           20: //включаем ПИД ДВ (если режим работы от ПЧ)
               IF "DV_invertor_mode".Value THEN
                   IF "Control_DV".Mode = TRUE AND
                       "Control_DV".Mode_from_PLC = TRUE AND
                       "Control_DV".SP_PID = "RegMap".P_air_ventilation THEN
                       "Timer".VENTILATION_temp_IN := FALSE;
                       "Technology".Regim_ventilation_step := 22;
                   ELSE
                       "Control_DV".Mode := TRUE;
                       "Control_DV".Mode_from_PLC := TRUE;
                       "Control_DV".SP_PID := "RegMap".P_air_ventilation;
                       //переход на следующий шаг
                       "Timer".VENTILATION_temp_IN := FALSE;
                       "Technology".Regim_ventilation_step := 21;
                   END_IF;
               ELSE
                   "Control_DS".Mode_from_PLC := FALSE;
                   //переход через шаг (без ожидания)
                   "Timer".VENTILATION_temp_IN := FALSE;
                   "Technology".Regim_ventilation_step := 22;
               END_IF;

           21: //Ожидаем 6 сек
               "Timer".VENTILATION_temp_PT := T#6s;
               "Timer".VENTILATION_temp_IN := TRUE;
               //переход на следующий шаг
               IF "Timer".VENTILATION_temp_Q THEN
                   "Timer".VENTILATION_temp_IN := FALSE;
                   "Technology".Regim_ventilation_step := 22;
               END_IF;

           22: //Проверям достижение параметров вентиляции и удержание их в течении заданного времени
               "Timer".VENTILATION_temp_PT := T_CONV(INT_TO_DINT("Technology".SP_TIME_Ventilation_start) * 1000);
               "Timer".VENTILATION_temp_IN := "NAV_middle".Value AND     //НАВ достигли среднего положения
               NOT "NAD_close".Value AND  //НАД не закрыты
               "P_air_burner".Value > ("RegMap".P_air_ventilation * (100 - "Technology".DB_P_air_ventilation)) / 100 AND//Давление воздуха перед горелкой в норме
               (NOT "P_air_before_burner_min".Value OR "Protections_BLOCK".P_air_before_burner_min) AND
               //"Sensors".dP_furnace_boiler.Value > ("RegMap".dP_furnace_ventilation * (100 + "Technology".DB_dP_furnace_ventilation))/100 AND //Разряжение в норме
               "dP_furnace_boiler".Value < ("RegMap".dP_furnace_ventilation * (100 - "Technology".DB_dP_furnace_ventilation)) / 100 AND
               (NOT "dP_furnace_boiler_min".Value OR "Protections_BLOCK".dP_in_furnance_min);
               //переход на следующий шаг
               IF "Timer".VENTILATION_temp_Q THEN
                   "Timer".VENTILATION_temp_IN := FALSE;
                   "Timer".VENTILATION_IN := FALSE;
                   "Timer".VENTILATION_R := TRUE;
                   "Timer".VENTILATION_PT := T_CONV(INT_TO_DINT("Technology".SP_TIME_Ventilation) * 1000);
                   "Technology".Regim_ventilation_step := 23;
               END_IF;

           23: //ВЕНТИЛЯЦИЯ
               "Message".VENTILATION_run := "NAV_middle".Value AND     //НАВ достигли среднего положения
               NOT "NAD_close".Value AND  //НАД не закрыты
               "P_air_burner".Value > ("RegMap".P_air_ventilation * (100 - "Technology".DB_P_air_ventilation)) / 100 AND//Давление воздуха перед горелкой в норме
               (NOT "P_air_before_burner_min".Value OR "Protections_BLOCK".P_air_before_burner_min) AND
               //"Sensors".dP_furnace_boiler.Value > ("RegMap".dP_furnace_ventilation * (100 + "Technology".DB_dP_furnace_ventilation))/100 AND //Разряжение в норме
               "dP_furnace_boiler".Value < ("RegMap".dP_furnace_ventilation * (100 - "Technology".DB_dP_furnace_ventilation)) / 100 AND
               (NOT "dP_furnace_boiler_min".Value OR "Protections_BLOCK".dP_in_furnance_min);

               "Message".VENTILATION_not := NOT "Message".VENTILATION_run;

               "Message".VENTILATION_alarm := "Warning".P_air_before_burner_min OR "Warning".dP_furnace_boiler_min;

               //Запускаем таймер вентиляции (время задается уставкой) с контролем параметров:
               "Timer".VENTILATION_IN := "Message".VENTILATION_run;
               "Timer".VENTILATION_R := "Message".VENTILATION_alarm;
               "Timer".VENTILATION_PT := T_CONV(INT_TO_DINT("Technology".SP_TIME_Ventilation) * 1000);

               //Если таймер вентиляции вышел или если вентиляцию уже проводилась, то вентиляция успешно проведена
               IF "Timer".VENTILATION_Q OR "Technology".Ventilation_conducted THEN
                   "Timer".VENTILATION_IN := FALSE;
                   "Message".VENTILATION_run := FALSE;
                   "Message".VENTILATION_not := FALSE;
                   "Message".VENTILATION_alarm := FALSE;
                   "Message".VENTILATION_ok := TRUE;
                   "Technology".Ventilation_conducted := TRUE;
                   //переходим далее
                   "Technology".Regim_ventilation_step := 25;
                   "Technology".Test_press_run := FALSE;
                   "Technology".Test_ignition_run := FALSE;
               END_IF;
               //если вентиляция не выполнена, то переход на ожидание повторной вентиляции
               IF "Message".VENTILATION_alarm THEN
                   "Timer".VENTILATION_IN := FALSE;
                   "Message".VENTILATION_run := FALSE;
                   "Message".VENTILATION_not := FALSE;
                   "Technology".Regim_ventilation_step := 24;
               END_IF;

           24: //ожидание повторной команды при неудачной вентиляции 
               //повторная вентиляция
               IF "Btn_Ventilation".Value OR
                   "FRONT".Btn_Ventilation_HMI OR
                   "FRONT".Btn_Ventilation_SCADA THEN
                   "Message".VENTILATION_alarm := FALSE;
                   "Technology".Regim_ventilation_step := 0;
               END_IF;

           25: //ожидание выхода из вентиляции
               //взводим защиту Понижение давления воздуха перед горелкой
               "Alarm_Enable".P_air_before_burner_min := TRUE;
               //взводим защиту Понижение разряжения в топке
               "Alarm_Enable".dP_furnace_boiler_min := TRUE;
               //Если нажата кнопка РОЗЖИГ
               IF ("Btn_Ignition".Value OR "FRONT".Btn_Ignition_HMI OR "FRONT".Btn_Ignition_SCADA) THEN
                   //сброс розжиговых предупреждений    
                   "Warning".Not_flame_Igniter := FALSE;
                   "Warning".PZK2_not_open := FALSE;

                   IF //и все параматры вентиляци в норме
                       "NAV_middle".Value AND     //НАВ достигли среднего положения
                       NOT "NAD_close".Value AND  //НАД не закрыты
                       "P_air_burner".Value > ("RegMap".P_air_ventilation * (100 - "Technology".DB_P_air_ventilation)) / 100 AND//Давление воздуха перед горелкой в норме
                       (NOT "P_air_before_burner_min".Value OR "Protections_BLOCK".P_air_before_burner_min) AND
                       //"Sensors".dP_furnace_boiler.Value > ("RegMap".dP_furnace_ventilation * (100 + "Technology".DB_dP_furnace_ventilation))/100 AND //Разряжение в норме
                       "dP_furnace_boiler".Value < ("RegMap".dP_furnace_ventilation * (100 - "Technology".DB_dP_furnace_ventilation)) / 100 AND
                       (NOT "dP_furnace_boiler_min".Value OR "Protections_BLOCK".dP_in_furnance_min) THEN
                       "Message".VENTILATION_Check_param := FALSE;
                       "Message".VENTILATION_ok := FALSE;
                       //переход на ОПРЕССОВКА
                       "Technology".Regim := 4;
                   ELSE
                       "Message".VENTILATION_Check_param := TRUE;
                   END_IF;
               END_IF;

               //переход на ТЕСТОВУЮ ОПРЕССОВКУ по нажатию на кн.ТЕСТОВАЯ ОПРЕССОВКА
               IF "FRONT".Btn_test_press_HMI THEN
                   //сброс розжиговых предупреждений    
                   "Warning".Not_flame_Igniter := FALSE;
                   "Warning".PZK2_not_open := FALSE;

                   IF //и все параматры вентиляци в норме
                       "NAV_middle".Value AND     //НАВ достигли среднего положения
                       NOT "NAD_close".Value AND  //НАД не закрыты
                       "P_air_burner".Value > ("RegMap".P_air_ventilation * (100 - "Technology".DB_P_air_ventilation)) / 100 AND//Давление воздуха перед горелкой в норме
                       (NOT "P_air_before_burner_min".Value OR "Protections_BLOCK".P_air_before_burner_min) AND
                       //"Sensors".dP_furnace_boiler.Value > ("RegMap".dP_furnace_ventilation * (100 + "Technology".DB_dP_furnace_ventilation))/100 AND //Разряжение в норме
                       "dP_furnace_boiler".Value < ("RegMap".dP_furnace_ventilation * (100 - "Technology".DB_dP_furnace_ventilation)) / 100 AND
                       (NOT "dP_furnace_boiler_min".Value OR "Protections_BLOCK".dP_in_furnance_min) THEN
                       "Message".VENTILATION_Check_param := FALSE;
                       "Message".VENTILATION_ok := FALSE;
                       //переход на ТЕСТОВАЯ ОПРЕССОВКА (ОПРЕССОВКА с 6 шага)                   
                       "Technology".Regim := 4;
                       "Technology".Regim_press_step := 6;
                       "Technology".Test_press_run := TRUE;
                       "Message".TEST_PRESS_ok := FALSE;
                   ELSE
                       "Message".VENTILATION_Check_param := TRUE;
                   END_IF;
               END_IF;

               //переход на ТЕСТОВЫЙ РОЗЖИГ по нажатию на кн.ТЕСТОВЫЙ РОЗЖИГ
               IF "FRONT".Btn_test_ignition_HMI THEN
                   //сброс розжиговых предупреждений    
                   "Warning".Not_flame_Igniter := FALSE;
                   "Warning".PZK2_not_open := FALSE;

                   IF //и все параматры вентиляци в норме
                       "NAV_middle".Value AND     //НАВ достигли среднего положения
                       NOT "NAD_close".Value AND  //НАД не закрыты
                       "P_air_burner".Value > ("RegMap".P_air_ventilation * (100 - "Technology".DB_P_air_ventilation)) / 100 AND//Давление воздуха перед горелкой в норме
                       (NOT "P_air_before_burner_min".Value OR "Protections_BLOCK".P_air_before_burner_min) AND
                       //"Sensors".dP_furnace_boiler.Value > ("RegMap".dP_furnace_ventilation * (100 + "Technology".DB_dP_furnace_ventilation))/100 AND //Разряжение в норме
                       "dP_furnace_boiler".Value < ("RegMap".dP_furnace_ventilation * (100 - "Technology".DB_dP_furnace_ventilation)) / 100 AND
                       (NOT "dP_furnace_boiler_min".Value OR "Protections_BLOCK".dP_in_furnance_min) THEN
                       "Message".VENTILATION_Check_param := FALSE;
                       "Message".VENTILATION_ok := FALSE;
                       //переход на ТЕСТОВЫЙ РОЗЖИГ (РОЗЖИГ)                   
                       "Technology".Regim := 5;
                       "Technology".Test_ignition_run := TRUE;
                       "Message".TEST_IGNITION_ok := FALSE;
                       //открываем ЗДГ
                       "Control_ZDG".Mode := TRUE;
                       "Control_ZDG".Avto_open := TRUE;
                   ELSE
                       "Message".VENTILATION_Check_param := TRUE;
                   END_IF;
               END_IF;

               //переход на РУЧНОЙ РОЗЖИГ по гажатию на кн. РУЧНОЙ РОЗЖИГ
               IF "HMI".Btn_manual_ignition_HMI THEN
                   //сброс розжиговых предупреждений    
                   "Warning".Not_flame_Igniter := FALSE;
                   "Warning".PZK2_not_open := FALSE;

                   IF //и все параматры вентиляци в норме
                       "NAV_middle".Value AND     //НАВ достигли среднего положения
                       NOT "NAD_close".Value AND  //НАД не закрыты
                       "P_air_burner".Value > ("RegMap".P_air_ventilation * (100 - "Technology".DB_P_air_ventilation)) / 100 AND//Давление воздуха перед горелкой в норме
                       (NOT "P_air_before_burner_min".Value OR "Protections_BLOCK".P_air_before_burner_min) AND
                       //"Sensors".dP_furnace_boiler.Value > ("RegMap".dP_furnace_ventilation * (100 + "Technology".DB_dP_furnace_ventilation))/100 AND //Разряжение в норме
                       "dP_furnace_boiler".Value < ("RegMap".dP_furnace_ventilation * (100 - "Technology".DB_dP_furnace_ventilation)) / 100 AND
                       (NOT "dP_furnace_boiler_min".Value OR "Protections_BLOCK".dP_in_furnance_min) THEN
                       "Message".VENTILATION_Check_param := FALSE;
                       "Message".VENTILATION_ok := FALSE;
                       //переход на РУЧНОЙ РОЗЖИГ                   
                       "Technology".Regim := 5;
                       "Technology".Regim_ignition_step := 19;
                       //открываем ЗДГ
                       "Control_ZDG".Mode := TRUE;
                       "Control_ZDG".Avto_open := TRUE;
                   ELSE
                       "Message".VENTILATION_Check_param := TRUE;
                   END_IF;
               END_IF;

           ELSE
               "Technology".Regim_ventilation_step := 0;
       END_CASE;
   ELSE
       //сброс текущего шага
       "Technology".Regim_ventilation_step := 0;
       //сброс сообщений
       "Message".VENTILATION_not_initial_state_gas := FALSE;
       "Message".VENTILATION_DS_need_dist_mode := FALSE;
       "Message".VENTILATION_DV_need_dist_mode := FALSE;
       "Message".VENTILATION_NAD_not_open := FALSE;
       "Message".VENTILATION_NAV_or_NAD_not_open := FALSE;
       "Message".VENTILATION_DS_not_on := FALSE;
       "Message".VENTILATION_DV_not_on := FALSE;
       "Message".VENTILATION_run := FALSE;
       "Message".VENTILATION_not := FALSE;
       "Message".VENTILATION_alarm := FALSE;
       "Message".VENTILATION_ok := FALSE;
       "Message".VENTILATION_Check_param := FALSE;
       "Message".VENTILATION_NAD_not_open_manual := FALSE;
       "Message".VENTILATION_NAV_not_open_manual := FALSE;
       "Message".VENTILATION_BRU_NAD_need_avto_mode := FALSE;
       "Message".VENTILATION_BRU_NAV_need_avto_mode := FALSE;
       //сброс таймеров
       "Timer".VENTILATION_temp_IN := FALSE;
       "Timer".VENTILATION_IN := FALSE;
       "Timer".VENTILATION_R := FALSE;
   END_IF;
END_FUNCTION

FUNCTION "Regim_OFF" : Void   // FC14, SCL
{ S7_Optimized_Access := 'TRUE' }
VERSION : 0.1
BEGIN
   (*Режим ОТКЛ*)
   (*таймеры*)
   (*процесс*)
   IF "Technology".Regim = 1 THEN
       CASE "Technology".Regim_off_step OF
           0:  // перевод управления всеми исполнительными устройствами в ручной режим
               "Control_ZRG".Mode:=FALSE;                  //ЗРГ
               "Control_ZRG".Mode_from_PLC := TRUE;
               "Control_ZDG".Mode:=FALSE;                  //ЗДГ
               "Control_ZDG".Avto_close := FALSE;
               "Control_ZDG".Avto_open := FALSE;
               "Control_ZDG".Avto_stop := FALSE;
               "Control_KB".Mode:=FALSE;                   //КБ
               "Control_KB".Avto_close := FALSE;
               "Control_KO".Mode:=FALSE;                   //КО
               "Control_KO".Avto_open := FALSE;
               "Control_KZ".Mode:=FALSE;                   //КЗ
               "Control_KZ".Avto_open := FALSE;
               "Control_PZK1".Mode:=FALSE;                 //ПЗК1
               "Control_PZK1".Avto_open := FALSE;
               "Control_PZK2".Mode:=FALSE;                 //ПЗК2
               "Control_PZK2".Avto_open := FALSE;
               "Control_IVN".Mode:=FALSE;                  //ИВН
               "Control_IVN".Avto_on := FALSE;
               "Control_ZDSV_before_boiler".Mode:=FALSE;   //ЗДСВ перед котлом
               "Control_ZDSV_before_boiler".Avto_close := FALSE;
               "Control_ZDSV_before_boiler".Avto_open := FALSE;
               "Control_ZDSV_before_boiler".Avto_stop := FALSE;
               "Control_GPZ".Mode := FALSE;                //ГПЗ
               "Control_GPZ".Avto_close := FALSE;
               "Control_GPZ".Avto_open := FALSE;
               "Control_GPZ".Avto_stop := FALSE;
               "Control_ZRW".Mode := FALSE;                //ЗРВ
               "Control_ZRW".Mode_from_PLC := TRUE;
               "Control_NAV".Mode:= FALSE;                 //НАВ
               "Control_NAV".Mode_from_PLC := TRUE;
               "Control_NAV".SP_PID := "RegMap".P_air_regim_map;
               "Control_NAV".Manual_close_from_PLC := FALSE;
               "Control_NAV".Manual_open_from_PLC := FALSE;
               "Control_NAD".Mode:= FALSE;                 //НАД
               "Control_NAD".Mode_from_PLC := TRUE;
               "Control_NAD".SP_PID := "RegMap".dP_furnace_regim_map;
               "Control_NAD".Manual_close_from_PLC := FALSE;
               "Control_NAD".Manual_open_from_PLC := FALSE;
               "Control_DV".Mode:= FALSE;                  //ДВ
               "Control_DV".Mode_from_PLC := TRUE;
               "Control_DV".SP_PID := "RegMap".P_air_regim_map;
               "Control_DV".Avto_Start := FALSE;
               "Control_DV".Avto_Stop := FALSE;
               "Control_DS".Mode:= FALSE;                  //ДС
               "Control_DS".Mode_from_PLC := TRUE;
               "Control_DS".SP_PID := "RegMap".dP_furnace_regim_map;
               "Control_DS".Avto_Start := FALSE;
               "Control_DS".Avto_Stop := FALSE;

           1:   //Ничего не делаем
               ;

           2:  //перевод всех клапанов в исходное состояние
               //все газовые клапана переводим в исходное состояние
               "Control_PZK1".Mode := TRUE;    //закрываем ПЗК1
               "Control_PZK1".Avto_open := FALSE;
               "Control_PZK2".Mode := TRUE;    //закрываем ПЗК2
               "Control_PZK2".Avto_open := FALSE;
               "Control_KO".Mode := TRUE;  //закрываем КО
               "Control_KO".Avto_open := FALSE;
               "Control_KZ".Mode := TRUE;  //закрываем КЗ
               "Control_KZ".Avto_open := FALSE;
               "Control_KB".Mode := TRUE;  //открываем КБ
               "Control_KB".Avto_close := FALSE;
               "Control_IVN".Mode := TRUE; //отключаем ИВН
               "Control_IVN".Avto_on := FALSE;

               "Control_ZRG".Mode := FALSE;                  //ЗРГ
               "Control_ZRG".Mode_from_PLC := TRUE;

               //контроль положения клапанов
               IF NOT "PZK1_open".Value AND
                   NOT "PZK2_not_close".Value AND
                   NOT "KO_open".Value AND
                   NOT "KZ_open".Value AND
                   NOT "KB_close".Value THEN
                   "Technology".Regim_off_step := 3;
               END_IF;

           3:  //снимаем защиту Отключение ДВ
               "Alarm_Enable".DV_off := FALSE;
               //отключение ДВ
               "Control_DV".Mode := TRUE;
               "Control_DV".Mode_from_PLC := FALSE;
               "Control_DV".Avto_Stop := TRUE;
               IF NOT "DV_invertor_on".Value AND NOT "DV_powergrid_on".Value THEN
                   //переход на следующий шаг
                   "Technology".Regim_off_step := 4;
               END_IF;

           4: //снимаем защиту Отключение ДС
               "Alarm_Enable".DS_off := FALSE;
               //отключение ДС
               "Control_DS".Mode := TRUE;
               "Control_DS".Mode_from_PLC := FALSE;
               "Control_DS".Avto_Stop := TRUE;
               IF NOT "DS_invertor_on".Value AND NOT "DS_powergrid_on".Value THEN
                   "Technology".Regim_off_step := 0;
               END_IF;
           ELSE
               "Technology".Regim_off_step := 0;
       END_CASE;

       //нажатие кнопки ПЛАНОВЫЙ ОСТАНОВ
       IF "FRONT".Btn_Normal_stop_HMI OR
           "FRONT".Btn_Normal_stop_SCADA OR
           "FRONT".Btn_Alarm_stop_HMI OR
           "FRONT".Btn_Alarm_stop_SCADA THEN
           "Technology".Regim_off_step := 2;
       END_IF;
       //нажатие кнопки ВЕНТИЛЯЦИЯ
       IF "Btn_Ventilation".Value OR
           "FRONT".Btn_Ventilation_HMI OR
           "FRONT".Btn_Ventilation_SCADA THEN
           "Message".OFF_Waiting_btn_ventilation := FALSE;
           "Technology".Regim := 3;    //переход на вентиляцию
           "Message".VENTILATION_not_initial_state_air := FALSE;
           "Message".VENTILATION_NAV_not_close := FALSE;
       ELSE
           "Message".OFF_Waiting_btn_ventilation := TRUE;
       END_IF;

   ELSE
       //Сброс текущего шага
       "Technology".Regim_off_step := 0;
       //Сброс всех сообщений по данному режиму
       "Message".OFF_Waiting_btn_ventilation := FALSE;
       "Message".OFF_Param_ventilation_not_norm := FALSE;
       //сброс таймеров
   END_IF;
END_FUNCTION

FUNCTION "Regim_CHECK" : Void   // FC16, SCL
{ S7_Optimized_Access := 'TRUE' }
VERSION : 0.1
BEGIN
   (*Режим ПРОВЕРКА*)
   (*таймеры*)
   (*процесс*)
   IF "Technology".Regim = 2 THEN
       ;
   ELSE
       "Technology".Regim_check_step := 0;
   END_IF;
END_FUNCTION

FUNCTION "Regim_PRESS" : Void   // FC17, SCL
{ S7_Optimized_Access := 'TRUE' }
VERSION : 0.1
BEGIN
   (*Режим ОПРЕССОВКА*)
   (*таймеры*)
   "Timer_PRESS_temp_DB".TON(IN := "Timer".PRESS_temp_IN,
                                PT := "Timer".PRESS_temp_PT,
                                Q => "Timer".PRESS_temp_Q);
   (*процесс*)
   IF "Technology".Regim = 4 THEN
       CASE "Technology".Regim_press_step OF
           0:  //даем команду на полное открытие ЗДСВ и включение регулятора уровня
               "Control_ZDSV_before_boiler".Mode := TRUE;
               "Control_ZDSV_before_boiler".Avto_open := TRUE;
               "Control_ZRW".Mode := TRUE;
               "Control_ZRW".Mode_from_PLC := TRUE;
               //если ЗДВС перед котлом открыта и есть вода в барабане
               IF "ZDSV_before_boiler_no_close".Value AND (NOT "L_water_min".Value OR "Protections_BLOCK".L_water_min) THEN
                   //переходим на шаг 6
                   "Technology".Regim_press_step := 6;
               END_IF;

           1:  //перевод разрежения на розжиговые параметры
               //если режим работы ДС от сети, то регулируем ПИД НАД
               IF "DS_powergrid_mode".Value THEN
                   "Control_NAD".Mode := TRUE;
                   "Control_NAD".Mode_from_PLC := TRUE;
                   "Control_NAD".SP_PID := "RegMap".dP_furnace_ignition;
               END_IF;
               //если режим работы ДС от ПЧ, то регулируем ПИД ДС
               IF "DS_invertor_mode".Value THEN
                   "Control_DS".Mode := TRUE;
                   "Control_DS".Mode_from_PLC := TRUE;
                   "Control_DS".SP_PID := "RegMap".dP_furnace_ignition;
               END_IF;
               "Timer".PRESS_temp_IN := FALSE;
               //переход на следующий шаг
               "Technology".Regim_press_step := 2;

           2:  //Ожидаем 5 сек
               "Timer".PRESS_temp_PT := T#5s;
               "Timer".PRESS_temp_IN := TRUE;
               //переход на следующий шаг
               IF "Timer".PRESS_temp_Q THEN
                   "Timer".PRESS_temp_IN := FALSE;
                   "Technology".Regim_press_step := 3;
               END_IF;

           3:  //перевод давления воздуха на розжиговые параметры
               //если режим работы ДВ от сети, то регулируем ПИД НАВ
               IF "DV_powergrid_mode".Value THEN
                   "Control_NAV".Mode := TRUE;
                   "Control_NAV".Mode_from_PLC := TRUE;
                   "Control_NAV".SP_PID := "RegMap".P_air_ignition;
               END_IF;
               //если режим работы ДВ от ПЧ, то регулируем ПИД ДВ
               IF "DV_invertor_mode".Value THEN
                   "Control_DV".Mode := TRUE;
                   "Control_DV".Mode_from_PLC := TRUE;
                   "Control_DV".SP_PID := "RegMap".P_air_ignition;
               END_IF;
               "Timer".PRESS_temp_IN := FALSE;
               //IF ("P_air_burner".Value > ("RegMap".P_air_ventilation * (100 - "Technology".DB_P_air_ventilation)) / 100) AND
               //    ("P_air_burner".Value < ("RegMap".P_air_ventilation * (100 + "Technology".DB_P_air_ventilation)) / 100) THEN
                   //переход на следующий шаг
                   "Technology".Regim_press_step := 4;
               //END_IF;

           4:  //Ожидаем 5 сек
               "Timer".PRESS_temp_PT := T#5s;
               "Timer".PRESS_temp_IN := TRUE;
               //переход на следующий шаг
               IF "Timer".PRESS_temp_Q THEN
                   "Timer".PRESS_temp_IN := FALSE;
                   "Technology".Regim_press_step := 5;
               END_IF;

           5:  //проверка достижения розжиговых параметров в течении 10 секунд
               "Timer".PRESS_temp_PT := T#10s;
               "Timer".PRESS_temp_IN := "P_air_burner".Value > ("RegMap".P_air_ignition * (100 - "Technology".DB_P_air_ignition)) / 100 AND //Давление воздуха перед горелкой в норме
                                        "P_air_burner".Value < ("RegMap".P_air_ignition * (100 + "Technology".DB_P_air_ignition)) / 100 AND
               //"Sensors".dP_furnace_boiler.Value > ("RegMap".dP_furnace_ignition * (100 + "Technology".DB_dP_furnace_ignition))/100 AND //Разряжение в норме
               "dP_furnace_boiler".Value < ("RegMap".dP_furnace_ignition * (100 - "Technology".DB_dP_furnace_ignition))/100;
               IF "Timer".PRESS_temp_Q THEN
                   //переход на следующий шаг
                   "Timer".PRESS_temp_IN := FALSE;
                   //"Technology".Regim_press_step := 6;       
                   "Technology".Regim := 5;    //переход на РОЗЖИГ
               END_IF;

           6:  //перевод клапанов по газу в исходное состояние
               "Control_PZK1".Mode := TRUE;        //закрываем ПЗК1
               "Control_PZK1".Avto_open := FALSE;
               "Control_PZK2".Mode := TRUE;        //закрываем ПЗК2
               "Control_PZK2".Avto_open := FALSE;
               "Control_KZ".Mode := TRUE;          //закрываем КЗ
               "Control_KZ".Avto_open := FALSE;
               "Control_KO".Mode := TRUE;          //закрываем КО
               "Control_KO".Avto_open := FALSE;
               "Control_KB".Mode := TRUE;          //открываем КБ
               "Control_KB".Avto_close := FALSE;
               "Control_IVN".Mode := TRUE;         //отключаем ИВН
               "Control_IVN".Avto_on := FALSE;
               //запускаем контрольный таймер
               "Timer".PRESS_temp_PT := T#60s;
               "Timer".PRESS_temp_IN := TRUE;
               //проверяем положение ИМ по газу
               IF NOT "KB_close".Value AND //КБ открыт
                   NOT "KZ_open".Value AND //КЗ закрыт
                   NOT "KO_open".Value AND //КО закрыт
                   NOT "PZK1_open".Value AND   //ПЗК1 закрыт
                   NOT "PZK2_not_close".Value THEN  //ПЗК2 закрыт
                   //переход далее
                   "Timer".PRESS_temp_IN := FALSE;
                   "Message".PRESS_not_initial_state_gas := FALSE;
                   "Technology".Regim_press_step := 7;
               END_IF;
               //если контрольное время вышло
               IF "Timer".PRESS_temp_Q THEN
                   "Message".PRESS_not_initial_state_gas := TRUE;
               END_IF;

           7:  //Закрываем ЗРГ
               "Control_ZRG".Mode := TRUE;
               "Control_ZRG".Mode_from_PLC := FALSE;
               "Control_ZRG".Manual_close_from_PLC := TRUE;
               //запускаем контрольный таймер
               "Timer".PRESS_temp_PT := T#60s;
               "Timer".PRESS_temp_IN := TRUE;
               //Проверка закрытия ЗРГ
               IF "ZRG_close".Value THEN
                   //переход далее
                   "Timer".PRESS_temp_IN := FALSE;
                   "Message".PRESS_ZRG_not_close := FALSE;
                   "Technology".Regim_press_step := 8;
               END_IF;
               //если контрольное время вышло
               IF "Timer".PRESS_temp_Q THEN
                   "Message".PRESS_ZRG_not_close := TRUE;
               END_IF;

           8:  //открываем ЗДГ
               "Control_ZDG".Mode := TRUE;
               "Control_ZDG".Avto_open := TRUE;
               //запускаем контрольный таймер
               "Timer".PRESS_temp_PT := T#60s;
               "Timer".PRESS_temp_IN := TRUE;
               //контроль открытия ЗДГ
               IF NOT "ZDG_no_open".Value THEN
                   //переход далее
                   "Timer".PRESS_temp_IN := FALSE;
                   "Message".PRESS_ZDG_not_open := FALSE;
                   "Technology".Regim_press_step := 9;
               END_IF;
               //если контрольное время вышло
               IF "Timer".PRESS_temp_Q THEN
                   "Message".PRESS_ZDG_not_open := TRUE;
               END_IF;

           9:  //Ожидаем 5 сек
               "Timer".PRESS_temp_PT := T#5s;
               "Timer".PRESS_temp_IN := TRUE;
               //переход на следующий шаг
               IF "Timer".PRESS_temp_Q THEN
                   "Timer".PRESS_temp_IN := FALSE;
                   "Technology".Regim_press_step := 10;
               END_IF;

           10:  //Контроль давления перед БГ
               IF (NOT "P_gas_before_BG_max".Value OR "Protections_BLOCK".P_gas_before_BG_max) AND (NOT "P_gas_before_BG_min".Value OR "Protections_BLOCK".P_gas_before_BG_min) THEN
                   //если давление в норме, то
                   //взводим защиту Повышение давления газа перед БГ
                   "Alarm_Enable".P_gas_before_BG_max := TRUE;
                   //взводим защиту Понижение давления газа перед БГ
                   "Alarm_Enable".P_gas_before_BG_min := TRUE;
                   //идем далее (через шаг)
                   "Technology".Regim_press_step := 12;
               ELSE
                   //если давление не в норме, то идем на ожидание повторного нажатия на кн РОЗЖИГ
                   "Message".PRESS_P_before_BG_alarm := TRUE;
                   "Technology".Regim_press_step := 11;
               END_IF;

           11: //ожидание повторного нажатия кн.РОЗЖИГ
               IF ("Btn_Ignition".Value OR "FRONT".Btn_Ignition_HMI OR "FRONT".Btn_Ignition_SCADA) THEN
                   "Message".PRESS_P_before_BG_alarm := FALSE;
                   "Technology".Regim_press_step := 10;
               END_IF;

           12: //Проверяем исходное состояние клапанов, ЗРГ и ЗДГ
               IF NOT "KB_close".Value AND         //КБ открыт
                   NOT "KZ_open".Value AND         //КЗ закрыт
                   NOT "KO_open".Value AND         //КО закрыт
                   NOT "PZK1_open".Value AND       //ПЗК1 закрыт
                   NOT "PZK2_open".Value AND       //ПЗК2 закрыт
                   "ZRG_close".Value AND           //ЗРГ закрыт
                   NOT "ZDG_no_open".Value THEN    //ЗДГ открыт
                   //проверяем давление между ПЗК в течении 3 секунд
                   "Timer".PRESS_temp_PT := T#3s;
                   "Timer".PRESS_temp_IN := TRUE;
                   IF "Timer".PRESS_temp_Q THEN
                       "Timer".PRESS_temp_IN := FALSE;
                       "Technology".Regim_press_step := 13;
                   ELSE
                       //если давление не в норме, то идем на ожидание повторного нажатия на кн РОЗЖИГ
                       IF "P_gas_between_PZK1_and_PZK2".Value > 0.09 THEN
                           "Message".PRESS_PZK1_or_KO_untight := TRUE;
                           "Timer".PRESS_temp_IN := FALSE;
                           "Technology".Regim_press_step := 22;
                       END_IF;
                   END_IF;
               ELSE
                   //клапана, ЗРГ, ЗДГ не в исходном состоянии
                   "Message".PRESS_not_initial_state_gas := TRUE;
                   "Timer".PRESS_temp_IN := FALSE;
                   "Technology".Regim_press_step := 22;
               END_IF;

           13: //проверка давления между ПЗК
               //закрываем КБ
               "Control_KB".Mode := TRUE;
               "Control_KB".Avto_close := TRUE;
               //проверяем давление между ПЗК
               "Timer".PRESS_temp_PT := T_CONV(INT_TO_DINT("Technology".SP_TIME_check_P_between_PZK) * 1000);
               "Timer".PRESS_temp_IN := TRUE;
               IF "Timer".PRESS_temp_Q THEN
                   "Timer".PRESS_temp_IN := FALSE;
                   //переход на следующий шаг
                   "Technology".Regim_press_step := 14;
               ELSE
                   //если давление не в норме, то идем на ожидание повторного нажатия на кн РОЗЖИГ
                   IF "P_gas_between_PZK1_and_PZK2".Value > 0.09 THEN
                       "Message".PRESS_PZK1_or_KO_untight := TRUE;
                       "Timer".PRESS_temp_IN := FALSE;
                       "Technology".Regim_press_step := 22;
                   END_IF;
               END_IF;

           14: //проверка на MIN
               //открываем КО
               "Control_KO".Mode := TRUE;
               "Control_KO".Avto_open := TRUE;
               "Timer".PRESS_temp_PT := T#3s;
               "Timer".PRESS_temp_IN := "KO_open".Value;
               IF "Timer".PRESS_temp_Q THEN
                   "Timer".PRESS_temp_IN := FALSE;
                   //закрываем КО
                   "Control_KO".Mode := TRUE;
                   "Control_KO".Avto_open := FALSE;
                   //переходим на следующий шаг
                   "Technology".Regim_press_step := 15;
               ELSE
                   //если давление не в норме, то идем на ожидание повторного нажатия на кн РОЗЖИГ
                   IF "P_gas_between_PZK1_and_PZK2".Value > "Technology".SP_P_between_PZK_check_max THEN
                       "Message".PRESS_Not_orifice_plate_or_PZK1_untight := TRUE;
                       "Timer".PRESS_temp_IN := FALSE;
                       "Technology".Regim_press_step := 22;
                   END_IF;
               END_IF;

           15: //проверка на MIN (продолжение)
               //если давление не в норме, то идем на ожидание повторного нажатия на кн РОЗЖИГ
               IF "P_gas_between_PZK1_and_PZK2".Value < "Technology".SP_P_between_PZK_check_min THEN
                   "Message".PRESS_PZK2_or_KB_untight := TRUE;
                   "Technology".Regim_press_step := 22;
               ELSE
                   "Timer".PRESS_temp_IN := FALSE;
                   //если давление в норме, то идем на следующий шаг
                   "Technology".Regim_press_step := 16;
               END_IF;

           16: //Ожидаем 2 сек
               "Timer".PRESS_temp_PT := T#2s;
               "Timer".PRESS_temp_IN := TRUE;
               //переход на следующий шаг
               IF "Timer".PRESS_temp_Q THEN
                   "Timer".PRESS_temp_IN := FALSE;
                   "Technology".Regim_press_step := 17;
               END_IF;

           17: //проверка на MAX
               //открываем КБ на 3 секунды
               "Control_KB".Mode := TRUE;
               "Control_KB".Avto_close := FALSE;
               "Timer".PRESS_temp_PT := T#5s;
               "Timer".PRESS_temp_IN := NOT "KB_close".Value;
               IF "Timer".PRESS_temp_Q THEN
                   "Timer".PRESS_temp_IN := FALSE;
                   //закрываем КБ
                   "Control_KB".Mode := TRUE;
                   "Control_KB".Avto_close := TRUE;
                   "Timer".PRESS_temp_IN := FALSE;
                   //переходим на следующий шаг
                   "Technology".Regim_press_step := 18;
               END_IF;

           18: //Ожидаем 2 сек
               "Timer".PRESS_temp_PT := T#2s;
               "Timer".PRESS_temp_IN := TRUE;
               //переход на следующий шаг
               IF "Timer".PRESS_temp_Q THEN
                   "Timer".PRESS_temp_IN := FALSE;
                   "Technology".Regim_press_step := 19;
               END_IF;

           19: //проверка на MAX (продолжение)
               //открываем КО на 25 секунд
               "Control_KO".Mode := TRUE;
               "Control_KO".Avto_open := TRUE;
               "Timer".PRESS_temp_PT := T#25s;
               "Timer".PRESS_temp_IN := "KO_open".Value;
               IF "Timer".PRESS_temp_Q THEN
                   "Timer".PRESS_temp_IN := FALSE;
                   //закрываем КO
                   "Control_KO".Mode := TRUE;
                   "Control_KO".Avto_open := FALSE;
                   //переходим на следующий шаг
                   "Technology".Regim_press_step := 20;
               END_IF;

           20: //проверка на MAX (продолжение)
               //проверяем давление на max в течении времени уствки
               "Timer".PRESS_temp_PT := T_CONV(INT_TO_DINT("Technology".SP_TIME_check_P_between_PZK) * 1000);
               "Timer".PRESS_temp_IN := TRUE;
               IF "Timer".PRESS_temp_Q THEN
                   "Timer".PRESS_temp_IN := FALSE;
                   //переход на следующий шаг
                   "Technology".Regim_press_step := 21;
               ELSE
                   //если давление не в норме (низкое), то идем на ожидание повторного нажатия на кн РОЗЖИГ
                   IF "P_gas_between_PZK1_and_PZK2".Value < "Technology".SP_P_between_PZK_check_max THEN
                       "Message".PRESS_PZK2_or_KB_untight := TRUE;
                       "Timer".PRESS_temp_IN := FALSE;
                       "Technology".Regim_press_step := 22;
                   END_IF;
               END_IF;

           21: //проверка на MAX (продолжение)
               //проверяем давление на min
               IF "P_gas_between_PZK1_and_PZK2".Value < "Technology".SP_P_between_PZK_check_min THEN
                   "Message".PRESS_PZK2_or_KB_untight := TRUE;
                   "Technology".Regim_press_step := 22;
               ELSE
                   //Если тестовая опрессовка
                   IF "Technology".Test_press_run THEN
                       "Message".TEST_PRESS_ok := TRUE;
                       //сброс режима тестовой опрессовки
                       "Technology".Test_press_run := FALSE;
                       //открываем КБ
                       "Control_KB".Mode := TRUE;
                       "Control_KB".Avto_close := FALSE;
                       //переход на ВЕНТИЛЯЦИЯ
                       "Technology".Regim := 3;
                       //сразу в конец вентиляции
                       "Technology".Regim_ventilation_step := 25;
                   ELSE
                       //иначе
                       //открываем КБ
                       "Control_KB".Mode := TRUE;
                       "Control_KB".Avto_close := FALSE;
                       //переход на розжиговые параметры
                       "Timer".PRESS_temp_IN := FALSE;
                       "Technology".Regim_press_step := 23;
                       //"Technology".Regim := 5;    //переход на РОЗЖИГ
                   END_IF;
               END_IF;

           22: //перевод клапанов в исходное состояние
               "Control_KB".Mode := TRUE;          //открываем КБ
               "Control_KB".Avto_close := FALSE;
               "Control_KZ".Mode := TRUE;          //закрываем КЗ
               "Control_KZ".Avto_open := FALSE;
               "Control_KO".Mode := TRUE;          //закрываем КО
               "Control_KO".Avto_open := FALSE;
               "Control_PZK1".Mode := TRUE;        //закрываем ПЗК1
               "Control_PZK1".Avto_open := FALSE;
               "Control_PZK2".Mode := TRUE;        //закрываем ПЗК2
               "Control_PZK2".Avto_open := FALSE;
               //ожидание повторного нажатия кн.РОЗЖИГ
               IF ("Btn_Ignition".Value OR "FRONT".Btn_Ignition_HMI OR "FRONT".Btn_Ignition_SCADA) THEN
                   "Message".PRESS_not_initial_state_gas := FALSE;
                   "Message".PRESS_PZK1_or_KO_untight := FALSE;
                   "Message".PRESS_Not_orifice_plate_or_PZK1_untight := FALSE;
                   "Message".PRESS_PZK2_or_KB_untight := FALSE;
                   "Technology".Regim_press_step := 6;
               END_IF;

           23:  //Ожидаем 5 сек
               "Timer".PRESS_temp_PT := T#5s;
               "Timer".PRESS_temp_IN := TRUE;
               //переход на следующий шаг
               IF "Timer".PRESS_temp_Q THEN
                   "Timer".PRESS_temp_IN := FALSE;
                   "Technology".Regim_press_step := 1;
               END_IF;

           ELSE
               "Technology".Regim_press_step := 0;
       END_CASE;

       //выход из тестовой опрессовки
       IF "Technology".Test_press_run THEN
           //если нажата кн. Вентиляция
           IF "Btn_Ventilation".Value OR
               "FRONT".Btn_Ventilation_HMI OR
               "FRONT".Btn_Ventilation_SCADA THEN
               //перевод клапанов по газу в исходное состояние
               "Control_PZK1".Mode := TRUE;        //закрываем ПЗК1
               "Control_PZK1".Avto_open := FALSE;
               "Control_PZK2".Mode := TRUE;        //закрываем ПЗК2
               "Control_PZK2".Avto_open := FALSE;
               "Control_KZ".Mode := TRUE;          //закрываем КЗ
               "Control_KZ".Avto_open := FALSE;
               "Control_KO".Mode := TRUE;          //закрываем КО
               "Control_KO".Avto_open := FALSE;
               "Control_KB".Mode := TRUE;          //открываем КБ
               "Control_KB".Avto_close := FALSE;
               "Control_IVN".Mode := TRUE;         //отключаем ИВН
               "Control_IVN".Avto_on := FALSE;
               //сброс режима тестовой опрессовки
               "Technology".Test_press_run := FALSE;
               //снимаем защиту Повышение давления газа перед БГ
               "Alarm_Enable".P_gas_before_BG_max := FALSE;
               //снимаем защиту Понижение давления газа перед БГ
               "Alarm_Enable".P_gas_before_BG_min := FALSE;

               //переход на ВЕНТИЛЯЦИЯ
               "Technology".Regim := 3;
               //если вентиляция топки проведена, то переходим сразу в конец вентиляции
               IF "Technology".Ventilation_conducted THEN
                   "Technology".Regim_ventilation_step := 25;
               END_IF;
           END_IF;
       END_IF;

   ELSE
       //сброс текущего шага
       "Technology".Regim_press_step := 0;
       //сброс сообщений
       "Message".PRESS_not_initial_state_gas := FALSE;
       "Message".PRESS_ZRG_not_close := FALSE;
       "Message".PRESS_ZDG_not_open := FALSE;
       "Message".PRESS_P_before_BG_alarm := FALSE;
       "Message".PRESS_PZK1_or_KO_untight := FALSE;
       "Message".PRESS_Not_orifice_plate_or_PZK1_untight := FALSE;
       "Message".PRESS_PZK2_or_KB_untight := FALSE;
       //сброс таймеров
       "Timer".PRESS_temp_IN := FALSE;
   END_IF;
END_FUNCTION

FUNCTION "Regim_IGNITION" : Void   // FC18, SCL
{ S7_Optimized_Access := 'FALSE' }
VERSION : 0.1
BEGIN
   (*Режим РОЗЖИГ*)
   (*таймеры*)
   "Timer_IGNITION_temp_DB".TON(IN := "Timer".IGNITION_temp_IN,
                                PT := "Timer".IGNITION_temp_PT,
                                Q => "Timer".IGNITION_temp_Q);
   "Timer_IGNITION_control_flame_DB".TON(IN := "Timer".IGNITION_control_flame_IN,
                                         PT := "Timer".IGNITION_control_flame_PT,
                                         Q => "Timer".IGNITION_control_flame_Q);

   (*процесс*)
   IF "Technology".Regim = 5 THEN

       //взводим защиту Понижение уровня в барабане
       "Alarm_Enable".L_water_min := TRUE;
       //взводим защиту Повышение уровня в барабане
       "Alarm_Enable".L_water_max := TRUE;
       //взводим защиту Повышение давления в барабане
       "Alarm_Enable".P_steam_max := TRUE;

       CASE "Technology".Regim_ignition_step OF
           0:  //закрываем ЗРГ
               "Control_ZRG".Mode := TRUE;
               "Control_ZRG".Mode_from_PLC := FALSE;
               "Control_ZRG".Manual_close_from_PLC := TRUE;
               IF "ZRG_close".Value AND NOT "ZDG_no_open".Value THEN
                   "Message".IGNITION_ZRG_not_close := FALSE;
                   "Technology".Regim_ignition_step := 1;
                   //снимаем защиту Понижение давления воздуха перед горелкой
                   "Alarm_Enable".P_air_before_burner_min := FALSE;
                   //снимаем защиту Понижение разряжения в топке
                   "Alarm_Enable".dP_furnace_boiler_min := FALSE;
               ELSE
                   "Message".IGNITION_ZRG_not_close := TRUE;
               END_IF;

           1:  //контролируем закрытое положение ПЗК2
               IF NOT "PZK2_not_close".Value AND NOT "PZK2_open".Value THEN
                   "Message".IGNITION_PZK2_not_close := FALSE;
                   "Technology".Regim_ignition_step := 2;
               ELSE
                   "Message".IGNITION_PZK2_not_close := TRUE;
               END_IF;

           2:  //контролируем закрытое положение КЗ
               IF NOT "KZ_open".Value THEN
                   "Message".IGNITION_KZ_not_close := FALSE;
                   "Technology".Regim_ignition_step := 3;
               ELSE
                   "Message".IGNITION_KZ_not_close := TRUE;
               END_IF;

           3:  //закрываем КБ
               "Control_KB".Mode := TRUE;
               "Control_KB".Avto_close := TRUE;
               //запускаем контрольный таймер
               "Timer".IGNITION_temp_PT := T#5s;
               "Timer".IGNITION_temp_IN := TRUE;
               //проверяем положение KB
               IF "KB_close".Value THEN
                   "Timer".IGNITION_temp_IN := FALSE;
                   "Message".IGNITION_KB_not_close := FALSE;
                   "Technology".Regim_ignition_step := 4;
               END_IF;
               //если контрольное время вышло
               IF "Timer".IGNITION_temp_Q THEN
                   "Message".IGNITION_KB_not_close := TRUE;
               END_IF;

           4:  //задержка 1 сек
               "Timer".IGNITION_temp_PT := T#1s;
               "Timer".IGNITION_temp_IN := TRUE;
               //переход на следующий шаг
               IF "Timer".IGNITION_temp_Q THEN
                   "Timer".IGNITION_temp_IN := FALSE;
                   "Technology".Regim_ignition_step := 5;
               END_IF;

           5:  //открываем ПЗК1
               "Control_PZK1".Mode := TRUE;
               "Control_PZK1".Avto_open := TRUE;
               //запускаем контрольный таймер
               "Timer".IGNITION_temp_PT := T#5s;
               "Timer".IGNITION_temp_IN := TRUE;
               //проверяем положение ПЗК1
               IF "PZK1_open".Value THEN
                   "Technology".CNT_Igniter := 0;    //обнуляем счетчик попыток розжига запальника
                   "Timer".IGNITION_temp_IN := FALSE;
                   "Message".IGNITION_PZK1_not_open := FALSE;
                   "Technology".Regim_ignition_step := 6;
               END_IF;
               //если контрольное время вышло
               IF "Timer".IGNITION_temp_Q THEN
                   "Message".IGNITION_PZK1_not_open := TRUE;
               END_IF;

           6:  //задержка 5 сек
               "Timer".IGNITION_temp_PT := T#5s;
               "Timer".IGNITION_temp_IN := TRUE;
               //переход на следующий шаг
               IF "Timer".IGNITION_temp_Q THEN
                   "Timer".IGNITION_temp_IN := FALSE;
                   "Technology".Regim_ignition_step := 7;
               END_IF;

           7:  //включаем ИВН (на 6 секунд)
               "Control_IVN".Mode := TRUE;
               "Control_IVN".Avto_on := TRUE;
               "Timer".IGNITION_temp_IN := FALSE;
               "Technology".CNT_Igniter := "Technology".CNT_Igniter + 1;    //увеличиваем счетчик попыток розжига запальника
               "Technology".Regim_ignition_step := 8;

           8:  //задержка 1 сек
               "Timer".IGNITION_temp_PT := T#1s;
               "Timer".IGNITION_temp_IN := TRUE;
               //переход на следующий шаг
               IF "Timer".IGNITION_temp_Q THEN
                   "Timer".IGNITION_temp_IN := FALSE;
                   "Technology".Regim_ignition_step := 9;
               END_IF;

           9:  //открываем КЗ
               "Control_KZ".Mode := TRUE;
               "Control_KZ".Avto_open := TRUE;
               //запускаем контрольный таймер
               "Timer".IGNITION_temp_PT := T#2s;
               "Timer".IGNITION_temp_IN := TRUE;
               //проверяем положение КЗ
               IF "KZ_open".Value THEN
                   "Timer".IGNITION_temp_IN := FALSE;
                   "Message".IGNITION_KZ_not_open := FALSE;
                   "Technology".Regim_ignition_step := 10;
               END_IF;
               //если контрольное время вышло
               IF "Timer".IGNITION_temp_Q THEN
                   "Message".IGNITION_KZ_not_open := TRUE;
               END_IF;

           10:  //задержка 2 сек
               "Timer".IGNITION_temp_PT := T#2s;
               "Timer".IGNITION_temp_IN := TRUE;
               //переход на следующий шаг
               IF "Timer".IGNITION_temp_Q THEN
                   "Timer".IGNITION_temp_IN := FALSE;
                   "Timer".IGNITION_control_flame_IN := FALSE;
                   "Technology".Regim_ignition_step := 11;
               END_IF;

           11:  //контроль пламени запальника в течении 10 секунд
               "Timer".IGNITION_control_flame_PT := T#10s;
               "Timer".IGNITION_control_flame_IN := TRUE;
               //запальник успешно разжегся
               IF "Timer".IGNITION_control_flame_Q THEN
                   "Timer".IGNITION_control_flame_IN := FALSE;
                   //вводим контроль пламени запальника
                   "Warning_Enable".Not_flame_Igniter := TRUE;
                   //переход на следующий шаг
                   "Technology".Regim_ignition_step := 14;
               ELSE
                   //если запальник потух
                   IF NOT "Igniter_flame".Value THEN
                       //если была 1 попытка розжига
                       IF "Technology".CNT_Igniter = 1 THEN
                           //переход на 2 попытку розжига запальника
                           "Timer".IGNITION_control_flame_IN := FALSE;
                           "Technology".Regim_ignition_step := 20;
                           //если было более одной попытки розжига    
                       ELSE
                           "Timer".IGNITION_control_flame_IN := FALSE;
                           "Message".IGNITION_Not_flame_igniter := TRUE;
                           //переход на приведение клапанов в исходное состояние
                           "Technology".Regim_ignition_step := 12;
                       END_IF;
                   END_IF;
               END_IF;

           12: //перевод клапанов в исходное состояние
               "Control_PZK1".Mode := TRUE;    //закрываем ПЗК1
               "Control_PZK1".Avto_open := FALSE;
               "Control_PZK2".Mode := TRUE;    //закрываем ПЗК2
               "Control_PZK2".Avto_open := FALSE;
               "Control_KZ".Mode := TRUE;      //закрываем КЗ
               "Control_KZ".Avto_open := FALSE;
               "Control_KO".Mode := TRUE;      //закрываем КO
               "Control_KO".Avto_open := FALSE;
               "Control_KB".Mode := TRUE;      //открываем КБ
               "Control_KB".Avto_close := FALSE;
               "Control_IVN".Mode := true;     //отключаем ИВН
               "Control_IVN".Avto_on := FALSE;
               IF "Technology".Ventilation_conducted THEN
                   "Technology".Regim_ignition_step := 13;
               ELSE
                   //переход на ВЕНТИЛЯЦИЯ
                   "Technology".Regim := 3;
               END_IF;

           13: //ожидаем повторного нажатия кн РОЗЖИГ
               IF ("Btn_Ignition".Value OR "FRONT".Btn_Ignition_HMI OR "FRONT".Btn_Ignition_SCADA) THEN
                   //если все механизмы переведены в исходное состояние
                   IF NOT "PZK1_open".Value AND                                           //ПЗК1 закрыт
                       NOT "PZK2_not_close".Value AND NOT "PZK2_open".Value AND    //ПЗК2 закрыт
                       NOT "KZ_open".Value AND                                             //КЗ закрыт
                       NOT "KO_open".Value AND                                             //КO закрыт
                       NOT "KB_close".Value THEN                                            //КБ открыт
                       //переходим на повторный РОЗЖИГ
                       "Message".IGNITION_not_initial_state_gas := FALSE;
                       "Technology".Regim_ignition_step := 0;
                   ELSE
                       "Message".IGNITION_not_initial_state_gas := TRUE;
                   END_IF;
                   "Warning".Not_flame_Igniter := FALSE;
                   "Warning".PZK2_not_open := FALSE;
               END_IF;

           14: //открываем ПЗК2
               "Control_PZK2".Mode := TRUE;
               "Control_PZK2".Avto_open := TRUE;
               "Warning_Enable".PZK2_not_open := TRUE;   //вводим контроль времени открытия ПЗК2
               //запускаем отсчет времени закрытия запальника
               "Timer".close_KZ_IN := TRUE;
               //замораживаем ПИДЫ по разряжению
               "Control_NAD".Manual_close_from_PLC := FALSE;
               "Control_NAD".Manual_open_from_PLC := FALSE;
               "Control_NAD".Mode_from_PLC := FALSE;
               "Control_DS".Manual_frequency_from_PLC := "PID_analog_DS_DB".OUT;
               "Control_DS".Mode_from_PLC := FALSE;
               //замораживаем ПИДЫ по давлению воздуха
               "Control_NAV".Manual_close_from_PLC := FALSE;
               "Control_NAV".Manual_open_from_PLC := FALSE;
               "Control_NAV".Mode_from_PLC := FALSE;
               "Control_DV".Manual_frequency_from_PLC := "PID_analog_DV_DB".OUT;
               "Control_DV".Mode_from_PLC := FALSE;

               "Timer".IGNITION_temp_IN := FALSE;
               //переходим на следующий шаг
               "Technology".Regim_ignition_step := 15;

           15: //задержка 14 сек
               "Timer".IGNITION_temp_PT := T#14s;
               "Timer".IGNITION_temp_IN := TRUE;
               //переход на следующий шаг
               IF "Timer".IGNITION_temp_Q THEN
                   "Timer".IGNITION_temp_IN := FALSE;
                   "Technology".Regim_ignition_step := 16;
               END_IF;

           16: //снимаем контроль пламени запальника    
               "Warning_Enable".Not_flame_Igniter := FALSE;
               //вводим контроль пламени горелки
               "Alarm_Enable".Not_flame_burner := TRUE;
               "Message".IGNITION_Flame_burner_OK := TRUE;

               "Technology".Regim_ignition_step := 17;

           17: //ожидаем полного открытия ПЗК2
               IF "PZK2_open".Value THEN
                   //задержка 5 сек
                   "Timer".IGNITION_temp_PT := T#5s;
                   "Timer".IGNITION_temp_IN := TRUE;
                   //переход на следующий шаг
                   IF "Timer".IGNITION_temp_Q THEN
                       "Timer".IGNITION_temp_IN := FALSE;
                       "Message".IGNITION_Flame_burner_OK := FALSE;
                       //включаем ПИДЫ по разряжению
                       IF "DS_invertor_mode".Value THEN
                           "Control_DS".Mode_from_PLC := TRUE;
                       END_IF;
                       IF "DS_powergrid_mode".Value THEN
                           "Control_NAD".Mode_from_PLC := TRUE;
                       END_IF;
                       //включаем ПИДЫ по давлению воздуха
                       IF "DV_invertor_mode".Value THEN
                           "Control_DV".Mode_from_PLC := TRUE;
                       END_IF;
                       IF "DV_powergrid_mode".Value THEN
                           "Control_NAV".Mode_from_PLC := TRUE;
                       END_IF;
                       "Technology".Regim_ignition_step := 18;
                   END_IF;
               END_IF;


           18: //проверка закрытого положения КЗ
               IF NOT "KZ_control_open".Value THEN
                   //Если тестовый розжиг
                   IF "Technology".Test_ignition_run THEN
                       "Message".TEST_IGNITION_ok := TRUE;
                   ELSE
                       //иначе
                       //переход на ВЫХОД НА MIN МОЩНОСТЬ
                       "Technology".Regim := 6;
                   END_IF;
               END_IF;

           19: //режим РУЧНОЙ РОЗЖИГ
               //переводим в ручной режим
               (*КБ*)
               "Control_KB".Mode := FALSE;
               (*KO*)
               "Control_KO".Mode := FALSE;
               (*КЗ*)
               "Control_KZ".Mode := FALSE;
               (*ПЗК1*)
               "Control_PZK1".Mode := FALSE;
               (*ПЗК2*)
               "Control_PZK2".Mode := FALSE;
               (*ИВН*)
               "Control_IVN".Mode := FALSE;

               //если ПЗК2 открывается
               IF "PZK2_control_open".Value THEN
                   //замораживаем ПИДЫ по разряжению
                   "Control_NAD".Manual_close_from_PLC := FALSE;
                   "Control_NAD".Manual_open_from_PLC := FALSE;
                   "Control_NAD".Mode_from_PLC := FALSE;
                   "Control_DS".Manual_frequency_from_PLC := "PID_analog_DS_DB".OUT;
                   "Control_DS".Mode_from_PLC := FALSE;
                   //замораживаем ПИДЫ по давлению воздуха
                   "Control_NAV".Manual_close_from_PLC := FALSE;
                   "Control_NAV".Manual_open_from_PLC := FALSE;
                   "Control_NAV".Mode_from_PLC := FALSE;
                   "Control_DV".Manual_frequency_from_PLC := "PID_analog_DV_DB".OUT;
                   "Control_DV".Mode_from_PLC := FALSE;
               END_IF;
               //задержка 14 сек
               "Timer".IGNITION_temp_PT := T#14s;
               "Timer".IGNITION_temp_IN := "PZK2_control_open".Value;
               IF "Timer".IGNITION_temp_Q THEN
                   //вводим контроль пламени горелки
                   "Alarm_Enable".Not_flame_burner := TRUE;
               END_IF;
               //если ПЗК2 открыт
               IF "PZK2_open".Value AND "Timer".IGNITION_temp_Q THEN
                   //включаем ПИДЫ по разряжению
                   IF "DS_invertor_mode".Value THEN
                       "Control_DS".Mode_from_PLC := TRUE;
                   END_IF;
                   IF "DS_powergrid_mode".Value THEN
                       "Control_NAD".Mode_from_PLC := TRUE;
                   END_IF;
                   //включаем ПИДЫ по давлению воздуха
                   IF "DV_invertor_mode".Value THEN
                       "Control_DV".Mode_from_PLC := TRUE;
                   END_IF;
                   IF "DV_powergrid_mode".Value THEN
                       "Control_NAV".Mode_from_PLC := TRUE;
                   END_IF;
               END_IF;

               //если нажата кн. Вентиляция
               IF "Btn_Ventilation".Value OR "FRONT".Btn_Ventilation_HMI OR "FRONT".Btn_Ventilation_SCADA OR NOT "HMI".Btn_manual_ignition_HMI THEN
                   "HMI".Btn_manual_ignition_HMI := FALSE;
                   //снимаем контроль пламени горелки
                   "Alarm_Enable".Not_flame_burner := FALSE;
                   //перевод клапанов по газу в исходное состояние
                   "Control_PZK1".Mode := TRUE;        //закрываем ПЗК1
                   "Control_PZK1".Avto_open := FALSE;
                   "Control_PZK1".Manual_open := FALSE;
                   "Control_PZK2".Mode := TRUE;        //закрываем ПЗК2
                   "Control_PZK2".Avto_open := FALSE;
                   "Control_PZK2".Manual_open := FALSE;
                   "Control_KZ".Mode := TRUE;          //закрываем КЗ
                   "Control_KZ".Avto_open := FALSE;
                   "Control_KZ".Manual_open := FALSE;
                   "Control_KO".Mode := TRUE;          //закрываем КО
                   "Control_KO".Avto_open := FALSE;
                   "Control_KO".Manual_open := FALSE;
                   "Control_KB".Mode := TRUE;          //открываем КБ
                   "Control_KB".Avto_close := FALSE;
                   "Control_KB".Manual_close := FALSE;
                   "Control_IVN".Mode := TRUE;         //отключаем ИВН
                   "Control_IVN".Avto_on := FALSE;
                   "Control_IVN".Manual_on := FALSE;
                   //закрываем ЗДГ
                   "Control_ZDG".Mode := TRUE;
                   "Control_ZDG".Avto_close := TRUE;
                   "Control_ZDG".Avto_open := FALSE;
                   "Control_ZDG".Avto_stop := FALSE;
                   //включаем ПИДЫ по разряжению
                   IF "DS_invertor_mode".Value THEN
                       "Control_DS".Mode_from_PLC := TRUE;
                   END_IF;
                   IF "DS_powergrid_mode".Value THEN
                       "Control_NAD".Mode_from_PLC := TRUE;
                   END_IF;
                   //включаем ПИДЫ по давлению воздуха
                   IF "DV_invertor_mode".Value THEN
                       "Control_DV".Mode_from_PLC := TRUE;
                   END_IF;
                   IF "DV_powergrid_mode".Value THEN
                       "Control_NAV".Mode_from_PLC := TRUE;
                   END_IF;
                   "Timer".IGNITION_temp_IN := FALSE;
                   //переход на ВЕНТИЛЯЦИЯ
                   "Technology".Regim := 3;
                   //если вентиляция топки проведена, то переходим сразу в конец вентиляции
                   IF "Technology".Ventilation_conducted THEN
                       "Technology".Regim_ventilation_step := 25;
                   END_IF;
               END_IF;

           20: //закрываем КЗ и отключаем ИВН
               "Control_KZ".Mode := TRUE;
               "Control_KZ".Avto_open := FALSE;
               "Timer".close_KZ_IN := FALSE;
               "Control_IVN".Mode := TRUE;
               "Control_IVN".Avto_on := FALSE;
               IF NOT "KZ_open".Value AND NOT "IVN_control_on".Value THEN
                   "Technology".Regim_ignition_step := 21;
                   "Timer".IGNITION_temp_IN := FALSE;
               END_IF;

           21: //задержка 2 сек
               "Timer".IGNITION_temp_PT := T#2s;
               "Timer".IGNITION_temp_IN := TRUE;
               //переход на следующий шаг
               IF "Timer".IGNITION_temp_Q THEN
                   "Timer".IGNITION_temp_IN := FALSE;
                   "Technology".Regim_ignition_step := 7;
               END_IF;

           ELSE
               "Technology".Regim_ignition_step := 0;
       END_CASE;

       //выход из тестового розжига
       IF "Technology".Test_ignition_run THEN
           //если нажата кн. Вентиляция
           IF "Btn_Ventilation".Value OR "FRONT".Btn_Ventilation_HMI OR "FRONT".Btn_Ventilation_SCADA THEN
               //сброс режима тестового розжига
               "Technology".Test_ignition_run := FALSE;
               //снимаем контроль пламени горелки
               "Alarm_Enable".Not_flame_burner := FALSE;
               //перевод клапанов по газу в исходное состояние
               "Control_PZK1".Mode := TRUE;        //закрываем ПЗК1
               "Control_PZK1".Avto_open := FALSE;
               "Control_PZK2".Mode := TRUE;        //закрываем ПЗК2
               "Control_PZK2".Avto_open := FALSE;
               "Control_KZ".Mode := TRUE;          //закрываем КЗ
               "Control_KZ".Avto_open := FALSE;
               "Control_KO".Mode := TRUE;          //закрываем КО
               "Control_KO".Avto_open := FALSE;
               "Control_KB".Mode := TRUE;          //открываем КБ
               "Control_KB".Avto_close := FALSE;
               "Control_IVN".Mode := TRUE;         //отключаем ИВН
               "Control_IVN".Avto_on := FALSE;
               //закрываем ЗДГ
               "Control_ZDG".Mode := TRUE;
               "Control_ZDG".Avto_close := TRUE;
               "Control_ZDG".Avto_open := FALSE;
               "Control_ZDG".Avto_stop := FALSE;
               //переход на ВЕНТИЛЯЦИЯ
               "Technology".Regim := 3;
               //если вентиляция топки проведена, то переходим сразу в конец вентиляции
               IF "Technology".Ventilation_conducted THEN
                   "Technology".Regim_ventilation_step := 25;
               END_IF;
           END_IF;
       END_IF;

       //в случае погасания запальника или аварии ПЗК2
       IF ("Warning".Not_flame_Igniter AND "Warning_Enable".Not_flame_Igniter) OR ("Warning".PZK2_not_open AND "Warning_Enable".PZK2_not_open) THEN
           "Technology".Regim_ignition_step := 12;
           "Warning_Enable".Not_flame_Igniter := FALSE;
           "Warning_Enable".PZK2_not_open := FALSE;
       END_IF;
   ELSE
       //сброс текущего шага
       "Technology".Regim_ignition_step := 0;
       //сброс сообщений
       "Message".IGNITION_ZRG_not_close := FALSE;
       "Message".IGNITION_PZK2_not_close := FALSE;
       "Message".IGNITION_KZ_not_close := FALSE;
       "Message".IGNITION_KB_not_close := FALSE;
       "Message".IGNITION_PZK1_not_open := FALSE;
       "Message".IGNITION_KZ_not_open := FALSE;
       "Message".IGNITION_Not_flame_igniter := FALSE;
       "Message".IGNITION_not_initial_state_gas := FALSE;
       "Message".IGNITION_Flame_burner_OK := FALSE;
       //сброс таймеров
       "Timer".IGNITION_temp_IN := FALSE;
       "Timer".IGNITION_control_flame_IN := FALSE;
       //снимаем контроль пламени запальника    
       "Warning_Enable".Not_flame_Igniter := FALSE;
       //снимаем контроль времени открытия ПЗК2
       "Warning_Enable".PZK2_not_open := FALSE;
   END_IF;
END_FUNCTION

FUNCTION "Regim_EMERGENCY_STOP" : Void   // FC19, SCL
{ S7_Optimized_Access := 'TRUE' }
VERSION : 0.1
BEGIN
   (*Режим ЭКСТРЕННЫЙ ОСТАНОВ*)
   (*таймеры*)
   "Timer_EMERGENCY_STOP_temp_DB".TON(IN :="Timer".EMERGENCY_STOP_temp_IN,
                                      PT := "Timer".EMERGENCY_STOP_temp_PT,
                                      Q => "Timer".EMERGENCY_STOP_temp_Q);

   (*процесс*)
   IF "Technology".Regim = 9 THEN
       //снимаем защиту Понижение уровня в барабане
       "Alarm_Enable".L_water_min := FALSE;
       //снимаем защиту Повышение уровня в барабане
       "Alarm_Enable".L_water_max := FALSE;
       //снимаем защиту Повышение давления в барабане
       "Alarm_Enable".P_steam_max := FALSE;

       CASE "Technology".Regim_emergency_stop_step OF
           0:  //снимаем защиту Повышение давления газа перед БГ
               "Alarm_Enable".P_gas_before_BG_max := FALSE;
               //снимаем защиту Понижение давления газа перед БГ
               "Alarm_Enable".P_gas_before_BG_min := FALSE;
               //снимаем защиту Понижение давления газа перед горелкой
               "Alarm_Enable".P_gas_before_burner_min := FALSE;
               //снимаем защиту Повышение давления газа перед горелкой
               "Alarm_Enable".P_gas_before_burner_max := FALSE;
               //снимаем защиту Отключение ДС
               "Alarm_Enable".DS_off := FALSE;
               //снимаем защиту Отключение ДВ
               "Alarm_Enable".DV_off := FALSE;
               //снимаем защиту Понижение давления воздуха перед горелкой
               "Alarm_Enable".P_air_before_burner_min := FALSE;
               //снимаем защиту Понижение разряжения в топке
               "Alarm_Enable".dP_furnace_boiler_min := FALSE;
               //снимаем защиту Невоспламенение или погасание факела горелки котла
               "Alarm_Enable".Not_flame_burner := FALSE;

               //все клапана переводим в исходное состояние
               "Control_PZK1".Mode := TRUE;    //закрываем ПЗК1
               "Control_PZK1".Avto_open := FALSE;
               "Control_PZK2".Mode := TRUE;    //закрываем ПЗК2
               "Control_PZK2".Avto_open := FALSE;
               "Control_KO".Mode := TRUE;  //закрываем КО
               "Control_KO".Avto_open := FALSE;
               "Control_KZ".Mode := TRUE;  //закрываем КЗ
               "Control_KZ".Avto_open := FALSE;
               "Control_KB".Mode := TRUE;  //открываем КБ
               "Control_KB".Avto_close := FALSE;
               "Control_IVN".Mode := TRUE; //отключаем ИВН
               "Control_IVN".Avto_on := FALSE;
               "Control_ZDG".Mode := TRUE; //закрываем ЗДГ
               "Control_ZDG".Avto_open := FALSE;
               "Control_ZDG".Avto_stop := FALSE;
               "Control_ZDG".Avto_close := TRUE;
               "Control_DV".Mode := TRUE;  //отключаем ДВ
               "Control_DV".Mode_from_PLC := TRUE;
               "Control_DV".Avto_Start := FALSE;
               "Control_DV".Avto_Stop := TRUE;
               "Control_DS".Mode := TRUE;  //отключаем ДС
               "Control_DS".Mode_from_PLC := TRUE;
               "Control_DS".Avto_Start := FALSE;
               "Control_DS".Avto_Stop := TRUE;
               //отключаем ПИД регулирование ЗРГ
               "Control_ZRG".Mode_from_PLC := FALSE;
               "Control_ZRG".Manual_close_from_PLC := FALSE;
               "Control_ZRG".Manual_open_from_PLC := FALSE;

               //запускаем контрольный таймер
               "Timer".EMERGENCY_STOP_temp_PT := T#60s;
               "Timer".EMERGENCY_STOP_temp_IN := TRUE;

               //контроль положения клапанов, ЗДГ, состояния ДВ и ДС, отжатия кн. ОСТАНОВ
               IF NOT "PZK1_open".Value AND
                   NOT "PZK2_not_close".Value AND
                   NOT "KO_open".Value AND
                   NOT "KZ_open".Value AND
                   NOT "KB_close".Value AND
                   NOT "ZDG_no_close".Value AND
                   NOT "DV_invertor_on".Value AND
                   NOT "DV_powergrid_on".Value AND
                   NOT "DS_invertor_on".Value AND
                   NOT "DS_powergrid_on".Value AND
                   NOT "Btn_STOP".Value THEN

                   "Timer".EMERGENCY_STOP_temp_IN := FALSE;
                   "Message".EMERGENCY_STOP_not_initial_state := FALSE;
                   //переходим на режим ОТКЛ
                   "Technology".Regim := 1;
                   //перевод ГПЗ в автоматический режим управления
                   "Control_GPZ".Mode := TRUE;
               END_IF;
               //если контрольное время вышло
               IF "Timer".EMERGENCY_STOP_temp_Q THEN
                   "Message".EMERGENCY_STOP_not_initial_state := TRUE;
               END_IF;
           ELSE
               "Technology".Regim_emergency_stop_step := 0;
       END_CASE;
   ELSE
       //Сброс текущего шага
       "Technology".Regim_emergency_stop_step := 0;
       //Сброс всех сообщений по данному режиму
       "Message".EMERGENCY_STOP_not_initial_state := FALSE;
       //сброс таймеров
       "Timer".EMERGENCY_STOP_temp_IN := FALSE;
   END_IF;
END_FUNCTION

FUNCTION "Regim_ALARM_STOP" : Void   // FC20, SCL
{ S7_Optimized_Access := 'TRUE' }
VERSION : 0.1
BEGIN
   (*Режим АВАРИЙНЫЙ ОСТАНОВ*)
   (*таймеры*)
   "Timer_ALARM_STOP_temp_DB".TON(IN := "Timer".ALARM_STOP_temp_IN,
                                      PT := "Timer".ALARM_STOP_temp_PT,
                                      Q => "Timer".ALARM_STOP_temp_Q);

   (*процесс*)
       IF "Technology".Regim = 10 THEN

           //снимаем защиту Понижение уровня в барабане
           "Alarm_Enable".L_water_min := FALSE;
           //снимаем защиту Повышение уровня в барабане
           "Alarm_Enable".L_water_max := FALSE;
           //снимаем защиту Повышение давления в барабане
           "Alarm_Enable".P_steam_max := FALSE;

       CASE "Technology".Regim_alarm_stop_step OF
           0:  //снимаем защиту Понижение давления газа перед горелкой
               "Alarm_Enable".P_gas_before_burner_min := FALSE;
               //снимаем защиту Повышение давления газа перед горелкой
               "Alarm_Enable".P_gas_before_burner_max := FALSE;
               //снимаем защиту Невоспламенение или погасание факела горелки котла
               "Alarm_Enable".Not_flame_burner := FALSE;

               //все газовые клапана переводим в исходное состояние
               "Control_PZK1".Mode := TRUE;    //закрываем ПЗК1
               "Control_PZK1".Avto_open := FALSE;
               "Control_PZK2".Mode := TRUE;    //закрываем ПЗК2
               "Control_PZK2".Avto_open := FALSE;
               "Control_KO".Mode := TRUE;  //закрываем КО
               "Control_KO".Avto_open := FALSE;
               "Control_KZ".Mode := TRUE;  //закрываем КЗ
               "Control_KZ".Avto_open := FALSE;
               "Control_KB".Mode := TRUE;  //открываем КБ
               "Control_KB".Avto_close := FALSE;
               "Control_IVN".Mode := TRUE; //отключаем ИВН
               "Control_IVN".Avto_on := FALSE;
               //отключаем ПИД регулирование ЗРГ
               "Control_ZRG".Mode_from_PLC := FALSE;
               "Control_ZRG".Manual_close_from_PLC := FALSE;
               "Control_ZRG".Manual_open_from_PLC := FALSE;
               //запускаем контрольный таймер
               "Timer".ALARM_STOP_temp_PT := T#60s;
               "Timer".ALARM_STOP_temp_IN := TRUE;

               //перевод регуляторов разряжения и вентиляции на вентиляционные параметры
               IF "DS_invertor_mode".Value THEN
                   "Control_DS".Mode := TRUE;
                   "Control_DS".Mode_from_PLC := TRUE;
                   "Control_DS".SP_PID := "RegMap".dP_furnace_ventilation;
               END_IF;
               IF "DS_powergrid_mode".Value THEN
                   "Control_NAD".Mode := TRUE;
                   "Control_NAD".Mode_from_PLC := TRUE;
                   "Control_NAD".SP_PID := "RegMap".dP_furnace_ventilation;
               END_IF;
               IF "DV_invertor_mode".Value THEN
                   "Control_DV".Mode := TRUE;
                   "Control_DV".Mode_from_PLC := TRUE;
                   "Control_DV".SP_PID := "RegMap".P_air_ventilation;
               END_IF;
               IF "DV_powergrid_mode".Value THEN
                   "Control_NAV".Mode := TRUE;
                   "Control_NAV".Mode_from_PLC := TRUE;
                   "Control_NAV".SP_PID := "RegMap".P_air_ventilation;
               END_IF;

               //контроль положения клапанов
               IF NOT "PZK1_open".Value AND
                   NOT "PZK2_not_close".Value AND
                   NOT "KO_open".Value AND
                   NOT "KZ_open".Value AND
                   NOT "KB_close".Value THEN

                   "Timer".ALARM_STOP_temp_IN := FALSE;
                   "Message".ALARM_STOP_not_initial_state_gas := FALSE;
                   //переходим на режим ПОСТОСТАНОВОЧНУЮ ОПРЕССОВКУ
                   "Technology".Regim := 12;
                   //перевод ГПЗ в автоматический режим управления
                   "Control_GPZ".Mode := TRUE;
               END_IF;
               //если контрольное время вышло
               IF "Timer".ALARM_STOP_temp_Q THEN
                   "Message".ALARM_STOP_not_initial_state_gas := TRUE;
               END_IF;
           ELSE
               "Technology".Regim_alarm_stop_step := 0;
       END_CASE;
       (*защитное отключение ДВ и ДС*)
       //если не работает ДВ или ДС, то отключаем оба
       IF "Protections".DS_off THEN
           //снимаем защиту Отключение ДС
           "Alarm_Enable".DS_off := FALSE;
           //снимаем защиту Отключение ДВ
           "Alarm_Enable".DV_off := FALSE;
           //снимаем защиту Понижение давления воздуха перед горелкой
           "Alarm_Enable".P_air_before_burner_min := FALSE;
           //снимаем защиту Понижение разряжения в топке
           "Alarm_Enable".dP_furnace_boiler_min := FALSE;
           //отключаем ДВ
           "Control_DV".Mode := TRUE;
           "Control_DV".Avto_Start := FALSE;
           "Control_DV".Avto_Stop := TRUE;
           //отключаем ДC
           "Control_DS".Mode := TRUE;
           "Control_DS".Avto_Start := FALSE;
           "Control_DS".Avto_Stop := TRUE;
       END_IF;

       IF "Protections".DV_off THEN
           //снимаем защиту Отключение ДВ
           "Alarm_Enable".DV_off := FALSE;
           //снимаем защиту Понижение давления воздуха перед горелкой
           "Alarm_Enable".P_air_before_burner_min := FALSE;
           //отключаем ДВ
           "Control_DV".Mode := TRUE;
           "Control_DV".Avto_Start := FALSE;
           "Control_DV".Avto_Stop := TRUE;
       END_IF;

       IF "Protections".DS_off OR "Protections".DV_off THEN
           //все газовые клапана переводим в исходное состояние
           "Control_PZK1".Mode := TRUE;    //закрываем ПЗК1
           "Control_PZK1".Avto_open := FALSE;
           "Control_PZK2".Mode := TRUE;    //закрываем ПЗК2
           "Control_PZK2".Avto_open := FALSE;
           "Control_KO".Mode := TRUE;  //закрываем КО
           "Control_KO".Avto_open := FALSE;
           "Control_KZ".Mode := TRUE;  //закрываем КЗ
           "Control_KZ".Avto_open := FALSE;
           "Control_KB".Mode := TRUE;  //открываем КБ
           "Control_KB".Avto_close := FALSE;
           "Control_IVN".Mode := TRUE; //отключаем ИВН
           "Control_IVN".Avto_on := FALSE;

           //отключаем ПИД регулирование ЗРГ
           "Control_ZRG".Mode_from_PLC := FALSE;
           "Control_ZRG".Manual_close_from_PLC := FALSE;
           "Control_ZRG".Manual_open_from_PLC := FALSE;
       END_IF;

   ELSE
       //Сброс текущего шага
       "Technology".Regim_alarm_stop_step := 0;
       //Сброс всех сообщений по данному режиму
       "Message".ALARM_STOP_not_initial_state_gas := FALSE;
       //сброс таймеров
       "Timer".ALARM_STOP_temp_IN := FALSE;
   END_IF;
END_FUNCTION

FUNCTION "Regim_PLAN_STOP" : Void   // FC21, SCL
{ S7_Optimized_Access := 'TRUE' }
VERSION : 0.1
BEGIN
   (*Режим ПЛАНОВЫЙ ОСТАНОВ*)
   (*таймеры*)
   "Timer_PLAN_STOP_temp_DB".TON(IN := "Timer".PLAN_STOP_temp_IN,
                                  PT := "Timer".PLAN_STOP_temp_PT,
                                  Q => "Timer".PLAN_STOP_temp_Q);
   "Timer_STOP_MIN_POWER_1_DB".TON(IN := "Timer".STOP_MIN_POWER_1_IN,
                                    PT := "Timer".STOP_MIN_POWER_1_PT,
                                    Q => "Timer".STOP_MIN_POWER_1_Q);
   "Timer_STOP_MIN_POWER_2_DB".TON(IN := "Timer".STOP_MIN_POWER_2_IN,
                                    PT := "Timer".STOP_MIN_POWER_2_PT,
                                    Q => "Timer".STOP_MIN_POWER_2_Q);

    (*процесс*)
   IF "Technology".Regim = 11 THEN
       CASE "Technology".Regim_plan_stop_step OF
           0:  //импульсами закрываем ЗРГ до значения минимальной мощности
               "Control_ZRG".Mode := TRUE;
               "Control_ZRG".Mode_from_PLC := FALSE;

               IF "ZRG_middle".Value THEN
                   //выход на режим минимальной мощности
                   "Timer".STOP_MIN_POWER_1_PT := T_CONV(INT_TO_DINT("Technology".SP_TIME_MIN_power_ZRG_drive));
                   "Timer".STOP_MIN_POWER_2_PT := T_CONV(INT_TO_DINT("Technology".SP_TIME_MIN_power_ZRG_stop));
                   IF NOT "Timer".STOP_MIN_POWER_1_IN AND NOT "Timer".STOP_MIN_POWER_2_IN THEN
                       "Timer".STOP_MIN_POWER_1_IN := TRUE;
                   END_IF;
                   IF "Timer".STOP_MIN_POWER_1_Q THEN
                       "Timer".STOP_MIN_POWER_1_IN := FALSE;
                       "Timer".STOP_MIN_POWER_2_IN := TRUE;
                       "Control_ZRG".Manual_close_from_PLC := FALSE;
                   END_IF;
                   IF "Timer".STOP_MIN_POWER_2_Q THEN
                       "Timer".STOP_MIN_POWER_2_IN := FALSE;
                       "Timer".STOP_MIN_POWER_1_IN := TRUE;
                       "Control_ZRG".Manual_close_from_PLC := TRUE;
                   END_IF;

                   IF "DS_invertor_mode".Value THEN
                      "Control_DS".SP_PID := "RegMap".dP_furnace_regim_map;
                   END_IF;
                   IF "DS_powergrid_mode".Value THEN
                      "Control_NAD".SP_PID := "RegMap".dP_furnace_regim_map;
                   END_IF;
                   IF "DV_invertor_mode".Value THEN
                      "Control_DV".SP_PID := "RegMap".P_air_regim_map;
                   END_IF;
                   IF "DV_powergrid_mode".Value THEN
                      "Control_NAV".SP_PID := "RegMap".P_air_regim_map;
                   END_IF;
               ELSE
                   "Control_ZRG".Manual_close_from_PLC := FALSE;
                   //переход на следующий шаг
                   "Technology".Regim_plan_stop_step := 1;
               END_IF;

           1:  //Контроль достижения минимальной мощности
                   //снимаем защиту Понижение давления газа перед горелкой
                   "Alarm_Enable".P_gas_before_burner_min := FALSE;
                   //снимаем защиту Повышение давления газа перед горелкой
                   "Alarm_Enable".P_gas_before_burner_max := FALSE;
                   //отключаем ПИД регулирование ЗРГ
                   "Control_ZRG".Mode_from_PLC := FALSE;
                   "Control_ZRG".Manual_close_from_PLC := FALSE;
                   "Control_ZRG".Manual_open_from_PLC := FALSE;
                   //переход на следующий шаг
                   "Technology".Regim_plan_stop_step := 2;
                   //перевод ГПЗ в автоматический режим управления
                   "Control_GPZ".Mode := TRUE;

           2:  //снимаем защиту Понижение уровня в барабане
               "Alarm_Enable".L_water_min := FALSE;
               //снимаем защиту Повышение уровня в барабане
               "Alarm_Enable".L_water_max := FALSE;
               //снимаем защиту Повышение давления в барабане
               "Alarm_Enable".P_steam_max := FALSE;

               //снимаем защиту Невоспламенение или погасание факела горелки котла
               "Alarm_Enable".Not_flame_burner := FALSE;

               //перевод газовых исполнительных механизмов в исходное состояние
               "Control_PZK1".Mode := TRUE;    //закрываем ПЗК1
               "Control_PZK1".Avto_open := FALSE;
               "Control_PZK2".Mode := TRUE;    //закрываем ПЗК2
               "Control_PZK2".Avto_open := FALSE;
               "Control_KO".Mode := TRUE;  //закрываем КО
               "Control_KO".Avto_open := FALSE;
               "Control_KZ".Mode := TRUE;  //закрываем КЗ
               "Control_KZ".Avto_open := FALSE;
               "Control_KB".Mode := TRUE;  //открываем КБ
               "Control_KB".Avto_close := FALSE;
               "Control_IVN".Mode := TRUE; //отключаем ИВН
               "Control_IVN".Avto_on := FALSE;

               //перевод регуляторов разряжения и вентиляции на вентиляционные параметры
               IF "DS_invertor_mode".Value THEN
                   "Control_DS".Mode := TRUE;
                   "Control_DS".Mode_from_PLC := TRUE;
                   "Control_DS".SP_PID := "RegMap".dP_furnace_ventilation;
               END_IF;
               IF "DS_powergrid_mode".Value THEN
                   "Control_NAD".Mode := TRUE;
                   "Control_NAD".Mode_from_PLC := TRUE;
                   "Control_NAD".SP_PID := "RegMap".dP_furnace_ventilation;
               END_IF;
               IF "DV_invertor_mode".Value THEN
                   "Control_DV".Mode := TRUE;
                   "Control_DV".Mode_from_PLC := TRUE;
                   "Control_DV".SP_PID := "RegMap".P_air_ventilation;
               END_IF;
               IF "DV_powergrid_mode".Value THEN
                   "Control_NAV".Mode := TRUE;
                   "Control_NAV".Mode_from_PLC := TRUE;
                   "Control_NAV".SP_PID := "RegMap".P_air_ventilation;
               END_IF;

               //запускаем контрольный таймер
               "Timer".PLAN_STOP_temp_PT := T#60s;
               "Timer".PLAN_STOP_temp_IN := TRUE;
               //проверяем положение ИМ по газу
               IF NOT "PZK1_open".Value AND
                   NOT "PZK2_not_close".Value AND
                   NOT "KO_open".Value AND
                   NOT "KZ_open".Value AND
                   NOT "KB_close".Value THEN
                   //переход далее
                   "Timer".PLAN_STOP_temp_IN := FALSE;
                   "Message".PLAN_STOP_not_initial_state_gas := FALSE;
                   "Technology".Regim_plan_stop_step := 3;
               END_IF;
               //если контрольное время вышло
               IF "Timer".PLAN_STOP_temp_Q THEN
                   "Message".PLAN_STOP_not_initial_state_gas := TRUE;
               END_IF;

           3:  //задержка 6 сек
               "Timer".PLAN_STOP_temp_PT := T#6s;
               "Timer".PLAN_STOP_temp_IN := TRUE;
               //переход далее
               IF "Timer".PLAN_STOP_temp_Q THEN
                   "Timer".PLAN_STOP_temp_IN := FALSE;
                   //переход на режим ПОСТОСТАНОВОЧНАЯ ОПРЕССОВКА
                   "Technology".Regim := 12;
               END_IF;
           ELSE
               "Technology".Regim_plan_stop_step := 0;
       END_CASE;
   ELSE
       //Сброс текущего шага
       "Technology".Regim_plan_stop_step := 0;
       //Сброс всех сообщений по данному режиму
       "Message".PLAN_STOP_not_initial_state_gas := FALSE;
       //сброс таймеров
       "Timer".PLAN_STOP_temp_IN := FALSE;
       "Timer".STOP_MIN_POWER_1_IN := FALSE;
       "Timer".STOP_MIN_POWER_2_IN := FALSE;
   END_IF;
END_FUNCTION

FUNCTION "Regim_MIN_POWER" : Void   // FC22, SCL
{ S7_Optimized_Access := 'TRUE' }
VERSION : 0.1
BEGIN
   (*Режим ВЫХОД НА МИНИМАЛЬНУЮ МОЩНОСТЬ*)
   (*таймеры*)
   "Timer_MIN_POWER_temp_DB".TON(IN := "Timer".MIN_POWER_temp_IN,
                                PT := "Timer".MIN_POWER_temp_PT,
                                Q => "Timer".MIN_POWER_temp_Q);
   "Timer_MIN_POWER_1_DB".TON(IN := "Timer".MIN_POWER_1_IN,
                              PT := "Timer".MIN_POWER_1_PT,
                              Q => "Timer".MIN_POWER_1_Q);
   "Timer_MIN_POWER_2_DB".TON(IN := "Timer".MIN_POWER_2_IN,
                              PT := "Timer".MIN_POWER_2_PT,
                              Q => "Timer".MIN_POWER_2_Q);

   (*процесс*)
   IF "Technology".Regim = 6 THEN
       CASE "Technology".Regim_min_power_step OF
           0:  //переводим ПИД разряжения на работу по режимной карте
               //если работа от ПЧ
               IF "DS_invertor_mode".Value THEN
                   "Control_DS".Mode := TRUE;
                   "Control_DS".Mode_from_PLC := TRUE;
                   "Control_DS".SP_PID := "RegMap".dP_furnace_regim_map;
               END_IF;
               //если работа от сети
               IF "DS_powergrid_mode".Value THEN
                   "Control_NAD".Mode := TRUE;
                   "Control_NAD".Mode_from_PLC := TRUE;
                   "Control_NAD".SP_PID := "RegMap".dP_furnace_regim_map;
               END_IF;
               "Timer".MIN_POWER_temp_IN := FALSE;
               "Technology".Regim_min_power_step := 1;

           1:  //задержка 5 сек
               "Timer".MIN_POWER_temp_PT := T#5s;
               "Timer".MIN_POWER_temp_IN := TRUE;
               //переход на следующий шаг
               IF "Timer".MIN_POWER_temp_Q THEN
                   "Timer".MIN_POWER_temp_IN := FALSE;
                   "Technology".Regim_min_power_step := 2;
               END_IF;
               IF "DS_invertor_mode".Value THEN
                   "Control_DS".SP_PID := "RegMap".dP_furnace_regim_map;
               END_IF;
               IF "DS_powergrid_mode".Value THEN
                   "Control_NAD".SP_PID := "RegMap".dP_furnace_regim_map;
               END_IF;

           2:  //переводим ПИД давления воздуха на работу по режимной карте
               //если работа от ПЧ
               IF "DV_invertor_mode".Value THEN
                   "Control_DV".Mode := TRUE;
                   "Control_DV".Mode_from_PLC := TRUE;
                   "Control_DV".SP_PID := "RegMap".P_air_regim_map;
               END_IF;
               //если работа от сети
               IF "DV_powergrid_mode".Value THEN
                   "Control_NAV".Mode := TRUE;
                   "Control_NAV".Mode_from_PLC := TRUE;
                   "Control_NAV".SP_PID := "RegMap".P_air_regim_map;
               END_IF;
               "Technology".Regim_min_power_step := 3;

           3:  //задержка 5 сек
               "Timer".MIN_POWER_temp_PT := T#5s;
               "Timer".MIN_POWER_temp_IN := TRUE;
               //переход на следующий шаг
               IF "Timer".MIN_POWER_temp_Q THEN
                   "Timer".MIN_POWER_temp_IN := FALSE;
                   "Technology".Regim_min_power_step := 4;
               END_IF;
               IF "DS_invertor_mode".Value THEN
                   "Control_DS".SP_PID := "RegMap".dP_furnace_regim_map;
               END_IF;
               IF "DS_powergrid_mode".Value THEN
                   "Control_NAD".SP_PID := "RegMap".dP_furnace_regim_map;
               END_IF;
               IF "DV_invertor_mode".Value THEN
                   "Control_DV".SP_PID := "RegMap".P_air_regim_map;
               END_IF;
               IF "DV_powergrid_mode".Value THEN
                   "Control_NAV".SP_PID := "RegMap".P_air_regim_map;
               END_IF;

           4:  //импульсами открываем ЗРГ до значения минимальной мощности
               "Control_ZRG".Mode := TRUE;
               "Control_ZRG".Mode_from_PLC := FALSE;
               IF "DS_invertor_mode".Value THEN
                   "Control_DS".SP_PID := "RegMap".dP_furnace_regim_map;
               END_IF;
               IF "DS_powergrid_mode".Value THEN
                   "Control_NAD".SP_PID := "RegMap".dP_furnace_regim_map;
               END_IF;
               IF "DV_invertor_mode".Value THEN
                   "Control_DV".SP_PID := "RegMap".P_air_regim_map;
               END_IF;
               IF "DV_powergrid_mode".Value THEN
                   "Control_NAV".SP_PID := "RegMap".P_air_regim_map;
               END_IF;
               //достигнут режим минимальной мощности
               IF "ZRG_middle".Value THEN
                   "Control_ZRG".Manual_open_from_PLC := FALSE;
                   //взводим защиту Понижение давления газа перед горелкой
                   "Alarm_Enable".P_gas_before_burner_min := TRUE;
                   //взводим защиту Повышение давления газа перед горелкой
                   "Alarm_Enable".P_gas_before_burner_max := TRUE;
                   //взводим защиту Понижение давления воздуха перед горелкой
                   "Alarm_Enable".P_air_before_burner_min := TRUE;
                   //взводим защиту Понижение разряжения в топке
                   "Alarm_Enable".dP_furnace_boiler_min := TRUE;
                   //переходим на режим ПРОГРЕВ
                   "Technology".Regim := 7;
               ELSE
                   //выход на режим минимальной мощности
                   "Timer".MIN_POWER_1_PT := T_CONV(INT_TO_DINT("Technology".SP_TIME_MIN_power_ZRG_drive));
                   "Timer".MIN_POWER_2_PT := T_CONV(INT_TO_DINT("Technology".SP_TIME_MIN_power_ZRG_stop));
                   IF NOT "Timer".MIN_POWER_1_IN AND NOT "Timer".MIN_POWER_2_IN THEN
                       "Timer".MIN_POWER_1_IN := TRUE;
                   END_IF;
                   IF "Timer".MIN_POWER_1_Q THEN
                       "Timer".MIN_POWER_1_IN := FALSE;
                       "Timer".MIN_POWER_2_IN := TRUE;
                       "Control_ZRG".Manual_open_from_PLC := FALSE;
                   END_IF;
                   IF "Timer".MIN_POWER_2_Q THEN
                       "Timer".MIN_POWER_2_IN := FALSE;
                       "Timer".MIN_POWER_1_IN := TRUE;
                       "Control_ZRG".Manual_open_from_PLC := TRUE;
                   END_IF;
               END_IF;
           ELSE
               "Technology".Regim_min_power_step := 0;
       END_CASE;
   ELSE
       //сброс текущего шага
       "Technology".Regim_min_power_step := 0;
       //сброс сообщений
       //сброс таймеров
       "Timer".MIN_POWER_temp_IN := FALSE;
       "Timer".MIN_POWER_1_IN := FALSE;
       "Timer".MIN_POWER_2_IN := FALSE;
   END_IF;
END_FUNCTION

FUNCTION "Regim_HEATING" : Void   // FC23, SCL
{ S7_Optimized_Access := 'TRUE' }
VERSION : 0.1
BEGIN
   (*Режим ПРОГРЕВ*)
   (*таймеры*)
   "Timer_HEATING_temp_DB".TON(IN := "Timer".HEATING_temp_IN,
                               PT := "Timer".HEATING_temp_PT,
                               Q => "Timer".HEATING_temp_Q);

   (*процесс*)
   IF "Technology".Regim = 7 THEN
       CASE "Technology".Regim_heating_step OF
           0:  //переводим ЗРГ в дистанционный режим
               "Control_ZRG".Mode := FALSE;
               "Control_ZRG".Mode_from_PLC := TRUE;
               //анализ разрешения прогрева
               IF "Technology".Heating_enable THEN
                   //переход на следующий шаг
                   "Timer".HEATING_temp_IN := FALSE;
                   "Technology".Regim_heating_step := 1;
               ELSE
                   //переход на режим РАБОТА
                   "Technology".Regim := 8;
               END_IF;

           1:  //начинаем отсчет времени прогрева   
               "Timer".HEATING_temp_PT := T_CONV(INT_TO_DINT("Technology".SP_TIME_Heating) * 60000);
               "Timer".HEATING_temp_IN := TRUE;
               //если время прогрева вышло
               IF "Timer".HEATING_temp_Q THEN
                   "Timer".HEATING_temp_IN := FALSE;
                   //переходим в режим работа
                   "Technology".Regim := 8;
               END_IF;
           ELSE
               "Technology".Regim_heating_step := 0;
       END_CASE;
       IF "DS_invertor_mode".Value THEN
           "Control_DS".SP_PID := "RegMap".dP_furnace_regim_map;
       END_IF;
       IF "DS_powergrid_mode".Value THEN
           "Control_NAD".SP_PID := "RegMap".dP_furnace_regim_map;
       END_IF;
       IF "DV_invertor_mode".Value THEN
           "Control_DV".SP_PID := "RegMap".P_air_regim_map;
       END_IF;
       IF "DV_powergrid_mode".Value THEN
           "Control_NAV".SP_PID := "RegMap".P_air_regim_map;
       END_IF;
   ELSE
       //сброс текущего шага
       "Technology".Regim_heating_step := 0;
       //сброс сообщений
       //сброс таймеров
       "Timer".HEATING_temp_IN := FALSE;
   END_IF;
END_FUNCTION

FUNCTION "Regim_RUN" : Void   // FC24, SCL
{ S7_Optimized_Access := 'TRUE' }
VERSION : 0.1
BEGIN
   (*Режим РАБОТА*)
   (*таймеры*)
   "Timer".RUN_temp_PT := LT#106751d_23h_47m_16s_854ms_775us_807ns;
   "Timer_RUN_temp_DB".TON(IN := "Timer".RUN_temp_IN,
                           PT := "Timer".RUN_temp_PT,
                           Q => "Timer".RUN_temp_Q);

   (*процесс*)
   IF "Technology".Regim = 8 THEN
       "Timer".RUN_temp_IN := TRUE;
       CASE "Technology".Regim_run_step OF
           0:
               ;
           ELSE
               "Technology".Regim_run_step := 0;
       END_CASE;
       IF "DS_invertor_mode".Value THEN
           "Control_DS".SP_PID := "RegMap".dP_furnace_regim_map;
       END_IF;
       IF "DS_powergrid_mode".Value THEN
           "Control_NAD".SP_PID := "RegMap".dP_furnace_regim_map;
       END_IF;
       IF "DV_invertor_mode".Value THEN
           "Control_DV".SP_PID := "RegMap".P_air_regim_map;
       END_IF;
       IF "DV_powergrid_mode".Value THEN
           "Control_NAV".SP_PID := "RegMap".P_air_regim_map;
       END_IF;
   ELSE
       //сброс текущего шага
       "Technology".Regim_run_step := 0;
       //сброс сообщений
       //сброс таймеров
       "Timer".RUN_temp_IN := FALSE;
   END_IF;
END_FUNCTION

FUNCTION "Regim_STOP_PRESS" : Void   // FC26, SCL
{ S7_Optimized_Access := 'TRUE' }
VERSION : 0.1
BEGIN
   (*Режим ПОСТОСТАНОВОЧНАЯ ОПРЕССОВКА*)
   (*таймеры*)
   "Timer_STOP_PRESS_temp_DB".TON(IN := "Timer".STOP_PRESS_temp_IN,
                                  PT := "Timer".STOP_PRESS_temp_PT,
                                  Q => "Timer".STOP_PRESS_temp_Q);
   (*процесс*)
   IF "Technology".Regim = 12 THEN
       IF ("DV_invertor_on".Value OR "DV_powergrid_on".Value) AND
           ("DS_invertor_on".Value OR "DS_powergrid_on".Value) THEN
           CASE "Technology".Regim_stop_press_step OF
               0:  //анализ разрешения постостановочной опрессовки
                   IF "Technology".Stop_press_enable AND (NOT "Technology".Ventilation_conducted OR "Technology".transition_ignition) THEN
                       //переход на следующий шаг
                       "Technology".Regim_stop_press_step := 1;
                   ELSE
                       //переход на режим УКОРОЧЕННАЯ ВЕНТИЛЯЦИЯ
                       "Technology".Regim := 13;
                   END_IF;

               1:  //контроль положения исполнительных механизмов по газу
                   IF NOT "PZK1_open".Value AND
                       NOT "PZK2_not_close".Value AND
                       NOT "KO_open".Value AND
                       NOT "KZ_open".Value AND
                       NOT "KB_close".Value THEN
                       //переход на следующий шаг
                       "Technology".Regim_stop_press_step := 2;
                   END_IF;

               2:  //контроль min P 
                   IF "P_gas_between_PZK1_and_PZK2".Value < "Technology".SP_P_between_PZK_check_min THEN
                       //переход на следующий шаг
                       "Technology".Regim_stop_press_step := 3;
                   ELSE
                       "Message".STOP_PRESS_PZK1_or_KO_untight := TRUE;
                       "Technology".Regim_stop_press_step := 8;
                   END_IF;

               3:  //контроль max P
                   IF "P_gas_between_PZK1_and_PZK2".Value < "Technology".SP_P_between_PZK_check_max THEN
                       //переход на следующий шаг
                       "Technology".Regim_stop_press_step := 4;
                   ELSE
                       "Message".STOP_PRESS_PZK1_or_KO_untight := TRUE;
                       "Technology".Regim_stop_press_step := 8;
                   END_IF;

               4:  //закрываем КБ
                   "Control_KB".Mode := TRUE;
                   "Control_KB".Avto_close := TRUE;
                   //контроль положения
                   IF "KB_close".Value THEN
                       //переход на следующий шаг
                       "Timer".STOP_PRESS_temp_IN := FALSE;
                       "Technology".Regim_stop_press_step := 5;
                   END_IF;

               5:  //контроль отсутствия давления газа м/у ПЗК в течении заданного времени
                   "Timer".STOP_PRESS_temp_PT := T_CONV(INT_TO_DINT("Technology".SP_TIME_check_P_stop_press_min) * 1000);
                   "Timer".STOP_PRESS_temp_IN := TRUE;
                   IF "Timer".STOP_PRESS_temp_Q THEN
                       //переход на следующий шаг
                       "Timer".STOP_PRESS_temp_IN := FALSE;
                       "Technology".Regim_stop_press_step := 6;
                   ELSE
                       //если давление не в норме
                       IF ("P_gas_between_PZK1_and_PZK2".Value > "Technology".SP_P_between_PZK_check_min) OR
                           ("P_gas_between_PZK1_and_PZK2".Value > "Technology".SP_P_between_PZK_check_max) THEN
                           "Message".STOP_PRESS_PZK1_or_KO_untight := TRUE;
                           "Timer".STOP_PRESS_temp_IN := FALSE;
                           "Technology".Regim_stop_press_step := 8;
                       END_IF;
                   END_IF;

